// TIA Portal V17 export
// export: Created 2025-03-05T08:00:12.5882391Z, ExportSetting WithDefaults, DisplayName Totally Integrated Automation Portal, DisplayVersion V17 Update 8, DisplayName TIA Portal Openness, DisplayVersion V17 Update 8, DisplayName TIA Portal Version Control Interface, DisplayVersion V17, DisplayName SINAMICS Startdrive Advanced, DisplayVersion V17 SP2, DisplayName SINAMICS Startdrive G110M, G120, G120C, G120D, G120P, G115D, DisplayVersion V17 SP2, DisplayName SINAMICS Startdrive G130, G150, S120, S150, SINAMICS MV, S210, DisplayVersion V17 SP2, DisplayName STEP 7 Professional, DisplayVersion V17 Update 8, DisplayName SINUMERIK ONE STEP 7 Toolbox, DisplayVersion V17 Update 12, DisplayName SINUMERIK 840D sl STEP 7 Toolbox, DisplayVersion V17 Update 12, DisplayName STEP 7 Safety, DisplayVersion V17 Update 6, DisplayName WinCC Advanced, DisplayVersion V17 Update 8
FUNCTION "FC2121_MPP" : Void   // FC2121, LAD
{ S7_Optimized_Access := 'FALSE' }
AUTHOR : ETXETAR
VERSION : 1.0
// stored: AutoNumber false, IsIECCheckEnabled false, SetENOAutomatically false, UDAEnableTagReadback false
   VAR_TEMP
      ONE : Int;
      RETVAL1 : Int;
      SIMU_PANEL_HMI_SEL : Bool;   // SIMULATED PANEL IN HMI SELECTED
   END_VAR
   VAR CONSTANT
      FC_NUMBER : DInt := 2121;   // FC NUMBER
   END_VAR
   VAR_TEMP   // added for the SCL form of the ladder/FBD networks
      _w1 : Bool;
      _w2 : Bool;
   END_VAR
BEGIN

REGION Network 1: INPUTS
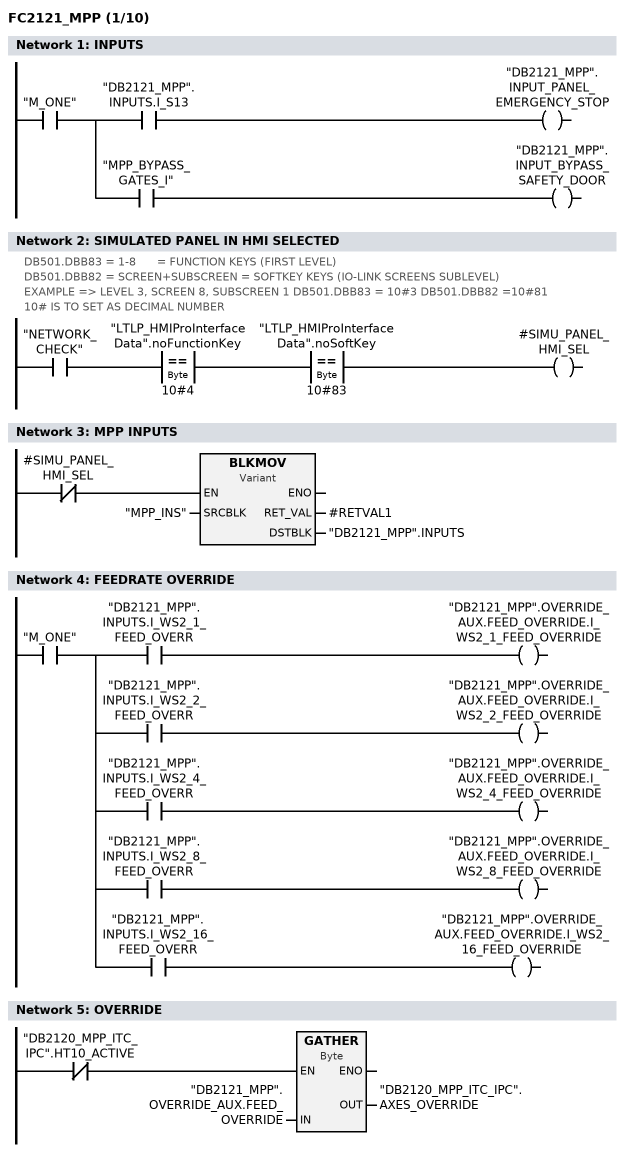
   RUNG wire#powerrail
      Contact( "M_ONE" )
      wire#w1
      Contact( "DB2121_MPP".INPUTS.I_S13 )
      Coil( "DB2121_MPP".INPUT_PANEL_EMERGENCY_STOP )
   END_RUNG
   RUNG wire#w1
      Contact( "MPP_BYPASS_GATES_I" )
      Coil( "DB2121_MPP".INPUT_BYPASS_SAFETY_DOOR )
   END_RUNG
   // the same network as SCL:
   "DB2121_MPP".INPUT_PANEL_EMERGENCY_STOP := "M_ONE" AND "DB2121_MPP".INPUTS.I_S13;
   "DB2121_MPP".INPUT_BYPASS_SAFETY_DOOR := "M_ONE" AND "MPP_BYPASS_GATES_I";
END_REGION

REGION Network 2: SIMULATED PANEL IN HMI SELECTED
   // DB501.DBB83 = 1-8      = FUNCTION KEYS (FIRST LEVEL)
   // DB501.DBB82 = SCREEN+SUBSCREEN = SOFTKEY KEYS (IO-LINK SCREENS SUBLEVEL)
   // EXAMPLE => LEVEL 3, SCREEN 8, SUBSCREEN 1 DB501.DBB83 = 10#3 DB501.DBB82 =10#81 
   // 10# IS TO SET AS DECIMAL NUMBER
   RUNG wire#powerrail
      Contact( "NETWORK_CHECK" )
      { S7_Templates := "SrcType := Byte" } EQ_Contact(in1 := "LTLP_HMIProInterfaceData".noFunctionKey, in2 := 10#4)
      { S7_Templates := "SrcType := Byte" } EQ_Contact(in1 := "LTLP_HMIProInterfaceData".noSoftKey, in2 := 10#83)
      Coil( #SIMU_PANEL_HMI_SEL )
   END_RUNG
   // the same network as SCL:
   #SIMU_PANEL_HMI_SEL := "NETWORK_CHECK" AND ("LTLP_HMIProInterfaceData".noFunctionKey = 10#4) AND ("LTLP_HMIProInterfaceData".noSoftKey = 10#83);
END_REGION

REGION Network 3: MPP INPUTS
   RUNG wire#powerrail
      I_Contact( #SIMU_PANEL_HMI_SEL )
      { S7_Templates := "blk_type := Variant" } BLKMOV(SRCBLK := "MPP_INS", RET_VAL => #RETVAL1, DSTBLK => "DB2121_MPP".INPUTS)
   END_RUNG
   // the same network as SCL:
   IF NOT #SIMU_PANEL_HMI_SEL THEN
       #RETVAL1 := BLKMOV(SRCBLK := "MPP_INS", DSTBLK => "DB2121_MPP".INPUTS);
   END_IF;
END_REGION

REGION Network 4: FEEDRATE OVERRIDE
   RUNG wire#powerrail
      Contact( "M_ONE" )
      wire#w1
      Contact( "DB2121_MPP".INPUTS.I_WS2_1_FEED_OVERR )
      Coil( "DB2121_MPP".OVERRIDE_AUX.FEED_OVERRIDE.I_WS2_1_FEED_OVERRIDE )
   END_RUNG
   RUNG wire#w1
      Contact( "DB2121_MPP".INPUTS.I_WS2_2_FEED_OVERR )
      Coil( "DB2121_MPP".OVERRIDE_AUX.FEED_OVERRIDE.I_WS2_2_FEED_OVERRIDE )
   END_RUNG
   RUNG wire#w1
      Contact( "DB2121_MPP".INPUTS.I_WS2_4_FEED_OVERR )
      Coil( "DB2121_MPP".OVERRIDE_AUX.FEED_OVERRIDE.I_WS2_4_FEED_OVERRIDE )
   END_RUNG
   RUNG wire#w1
      Contact( "DB2121_MPP".INPUTS.I_WS2_8_FEED_OVERR )
      Coil( "DB2121_MPP".OVERRIDE_AUX.FEED_OVERRIDE.I_WS2_8_FEED_OVERRIDE )
   END_RUNG
   RUNG wire#w1
      Contact( "DB2121_MPP".INPUTS.I_WS2_16_FEED_OVERR )
      Coil( "DB2121_MPP".OVERRIDE_AUX.FEED_OVERRIDE.I_WS2_16_FEED_OVERRIDE )
   END_RUNG
   // the same network as SCL:
   "DB2121_MPP".OVERRIDE_AUX.FEED_OVERRIDE.I_WS2_1_FEED_OVERRIDE := "M_ONE" AND "DB2121_MPP".INPUTS.I_WS2_1_FEED_OVERR;
   "DB2121_MPP".OVERRIDE_AUX.FEED_OVERRIDE.I_WS2_2_FEED_OVERRIDE := "M_ONE" AND "DB2121_MPP".INPUTS.I_WS2_2_FEED_OVERR;
   "DB2121_MPP".OVERRIDE_AUX.FEED_OVERRIDE.I_WS2_4_FEED_OVERRIDE := "M_ONE" AND "DB2121_MPP".INPUTS.I_WS2_4_FEED_OVERR;
   "DB2121_MPP".OVERRIDE_AUX.FEED_OVERRIDE.I_WS2_8_FEED_OVERRIDE := "M_ONE" AND "DB2121_MPP".INPUTS.I_WS2_8_FEED_OVERR;
   "DB2121_MPP".OVERRIDE_AUX.FEED_OVERRIDE.I_WS2_16_FEED_OVERRIDE := "M_ONE" AND "DB2121_MPP".INPUTS.I_WS2_16_FEED_OVERR;
END_REGION

REGION Network 5: OVERRIDE
   RUNG wire#powerrail
      I_Contact( "DB2120_MPP_ITC_IPC".HT10_ACTIVE )
      { S7_Templates := "[dest_type := Byte, src_type := Bool]" } GATHER(IN := "DB2121_MPP".OVERRIDE_AUX.FEED_OVERRIDE, OUT => "DB2120_MPP_ITC_IPC".AXES_OVERRIDE)
   END_RUNG
   // the same network as SCL:
   IF NOT "DB2120_MPP_ITC_IPC".HT10_ACTIVE THEN
       GATHER(IN := "DB2121_MPP".OVERRIDE_AUX.FEED_OVERRIDE, OUT => "DB2120_MPP_ITC_IPC".AXES_OVERRIDE);
   END_IF;
END_REGION

REGION Network 6: SPINDLES OVERRIDE
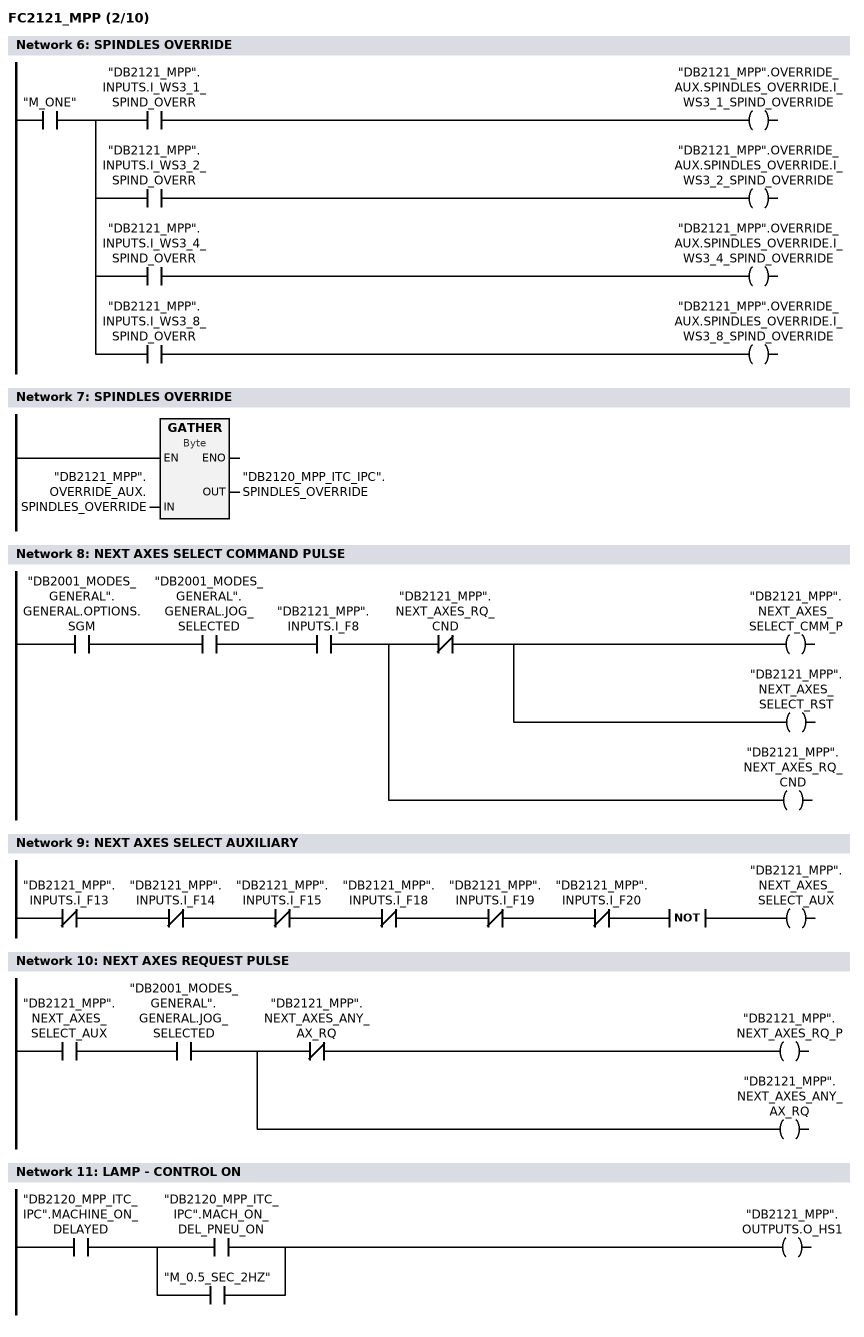
   RUNG wire#powerrail
      Contact( "M_ONE" )
      wire#w1
      Contact( "DB2121_MPP".INPUTS.I_WS3_1_SPIND_OVERR )
      Coil( "DB2121_MPP".OVERRIDE_AUX.SPINDLES_OVERRIDE.I_WS3_1_SPIND_OVERRIDE )
   END_RUNG
   RUNG wire#w1
      Contact( "DB2121_MPP".INPUTS.I_WS3_2_SPIND_OVERR )
      Coil( "DB2121_MPP".OVERRIDE_AUX.SPINDLES_OVERRIDE.I_WS3_2_SPIND_OVERRIDE )
   END_RUNG
   RUNG wire#w1
      Contact( "DB2121_MPP".INPUTS.I_WS3_4_SPIND_OVERR )
      Coil( "DB2121_MPP".OVERRIDE_AUX.SPINDLES_OVERRIDE.I_WS3_4_SPIND_OVERRIDE )
   END_RUNG
   RUNG wire#w1
      Contact( "DB2121_MPP".INPUTS.I_WS3_8_SPIND_OVERR )
      Coil( "DB2121_MPP".OVERRIDE_AUX.SPINDLES_OVERRIDE.I_WS3_8_SPIND_OVERRIDE )
   END_RUNG
   // the same network as SCL:
   "DB2121_MPP".OVERRIDE_AUX.SPINDLES_OVERRIDE.I_WS3_1_SPIND_OVERRIDE := "M_ONE" AND "DB2121_MPP".INPUTS.I_WS3_1_SPIND_OVERR;
   "DB2121_MPP".OVERRIDE_AUX.SPINDLES_OVERRIDE.I_WS3_2_SPIND_OVERRIDE := "M_ONE" AND "DB2121_MPP".INPUTS.I_WS3_2_SPIND_OVERR;
   "DB2121_MPP".OVERRIDE_AUX.SPINDLES_OVERRIDE.I_WS3_4_SPIND_OVERRIDE := "M_ONE" AND "DB2121_MPP".INPUTS.I_WS3_4_SPIND_OVERR;
   "DB2121_MPP".OVERRIDE_AUX.SPINDLES_OVERRIDE.I_WS3_8_SPIND_OVERRIDE := "M_ONE" AND "DB2121_MPP".INPUTS.I_WS3_8_SPIND_OVERR;
END_REGION

REGION Network 7: SPINDLES OVERRIDE
   RUNG wire#powerrail
      { S7_Templates := "[dest_type := Byte, src_type := Bool]" } GATHER(IN := "DB2121_MPP".OVERRIDE_AUX.SPINDLES_OVERRIDE, OUT => "DB2120_MPP_ITC_IPC".SPINDLES_OVERRIDE)
   END_RUNG
   // the same network as SCL:
   GATHER(IN := "DB2121_MPP".OVERRIDE_AUX.SPINDLES_OVERRIDE, OUT => "DB2120_MPP_ITC_IPC".SPINDLES_OVERRIDE);
END_REGION

REGION Network 8: NEXT AXES SELECT COMMAND PULSE
   RUNG wire#powerrail
      Contact( "DB2001_MODES_GENERAL".GENERAL.OPTIONS.SGM )
      Contact( "DB2001_MODES_GENERAL".GENERAL.JOG_SELECTED )
      Contact( "DB2121_MPP".INPUTS.I_F8 )
      wire#w1
      I_Contact( "DB2121_MPP".NEXT_AXES_RQ_CND )
      wire#w2
      Coil( "DB2121_MPP".NEXT_AXES_SELECT_CMM_P )
   END_RUNG
   RUNG wire#w2
      Coil( "DB2121_MPP".NEXT_AXES_SELECT_RST )
   END_RUNG
   RUNG wire#w1
      Coil( "DB2121_MPP".NEXT_AXES_RQ_CND )
   END_RUNG
   // the same network as SCL:
   #_w1 := "DB2001_MODES_GENERAL".GENERAL.OPTIONS.SGM AND "DB2001_MODES_GENERAL".GENERAL.JOG_SELECTED AND "DB2121_MPP".INPUTS.I_F8;
   "DB2121_MPP".NEXT_AXES_SELECT_CMM_P := #_w1 AND NOT "DB2121_MPP".NEXT_AXES_RQ_CND;
   "DB2121_MPP".NEXT_AXES_SELECT_RST := "DB2121_MPP".NEXT_AXES_SELECT_CMM_P;
   "DB2121_MPP".NEXT_AXES_RQ_CND := #_w1;
END_REGION

REGION Network 9: NEXT AXES SELECT AUXILIARY
   RUNG wire#powerrail
      I_Contact( "DB2121_MPP".INPUTS.I_F13 )
      I_Contact( "DB2121_MPP".INPUTS.I_F14 )
      I_Contact( "DB2121_MPP".INPUTS.I_F15 )
      I_Contact( "DB2121_MPP".INPUTS.I_F18 )
      I_Contact( "DB2121_MPP".INPUTS.I_F19 )
      I_Contact( "DB2121_MPP".INPUTS.I_F20 )
      Not()
      Coil( "DB2121_MPP".NEXT_AXES_SELECT_AUX )
   END_RUNG
   // the same network as SCL:
   "DB2121_MPP".NEXT_AXES_SELECT_AUX := NOT (NOT "DB2121_MPP".INPUTS.I_F13 AND NOT "DB2121_MPP".INPUTS.I_F14 AND NOT "DB2121_MPP".INPUTS.I_F15 AND NOT "DB2121_MPP".INPUTS.I_F18 AND NOT "DB2121_MPP".INPUTS.I_F19 AND NOT "DB2121_MPP".INPUTS.I_F20);
END_REGION

REGION Network 10: NEXT AXES REQUEST PULSE
   RUNG wire#powerrail
      Contact( "DB2121_MPP".NEXT_AXES_SELECT_AUX )
      Contact( "DB2001_MODES_GENERAL".GENERAL.JOG_SELECTED )
      wire#w1
      I_Contact( "DB2121_MPP".NEXT_AXES_ANY_AX_RQ )
      Coil( "DB2121_MPP".NEXT_AXES_RQ_P )
   END_RUNG
   RUNG wire#w1
      Coil( "DB2121_MPP".NEXT_AXES_ANY_AX_RQ )
   END_RUNG
   // the same network as SCL:
   #_w1 := "DB2121_MPP".NEXT_AXES_SELECT_AUX AND "DB2001_MODES_GENERAL".GENERAL.JOG_SELECTED;
   "DB2121_MPP".NEXT_AXES_RQ_P := #_w1 AND NOT "DB2121_MPP".NEXT_AXES_ANY_AX_RQ;
   "DB2121_MPP".NEXT_AXES_ANY_AX_RQ := #_w1;
END_REGION

REGION Network 11: LAMP - CONTROL ON
   RUNG wire#powerrail
      Contact( "DB2120_MPP_ITC_IPC".MACHINE_ON_DELAYED )
      wire#w1
      Contact( "DB2120_MPP_ITC_IPC".MACH_ON_DEL_PNEU_ON )
      wire#w2
      Coil( "DB2121_MPP".OUTPUTS.O_HS1 )
   END_RUNG
   RUNG wire#w1
      Contact( "M_0.5_SEC_2HZ" )
   END_RUNG wire#w2
   // the same network as SCL:
   "DB2121_MPP".OUTPUTS.O_HS1 := "DB2120_MPP_ITC_IPC".MACHINE_ON_DELAYED AND ("DB2120_MPP_ITC_IPC".MACH_ON_DEL_PNEU_ON OR "M_0.5_SEC_2HZ");
END_REGION

REGION Network 12: LAMP - HOME
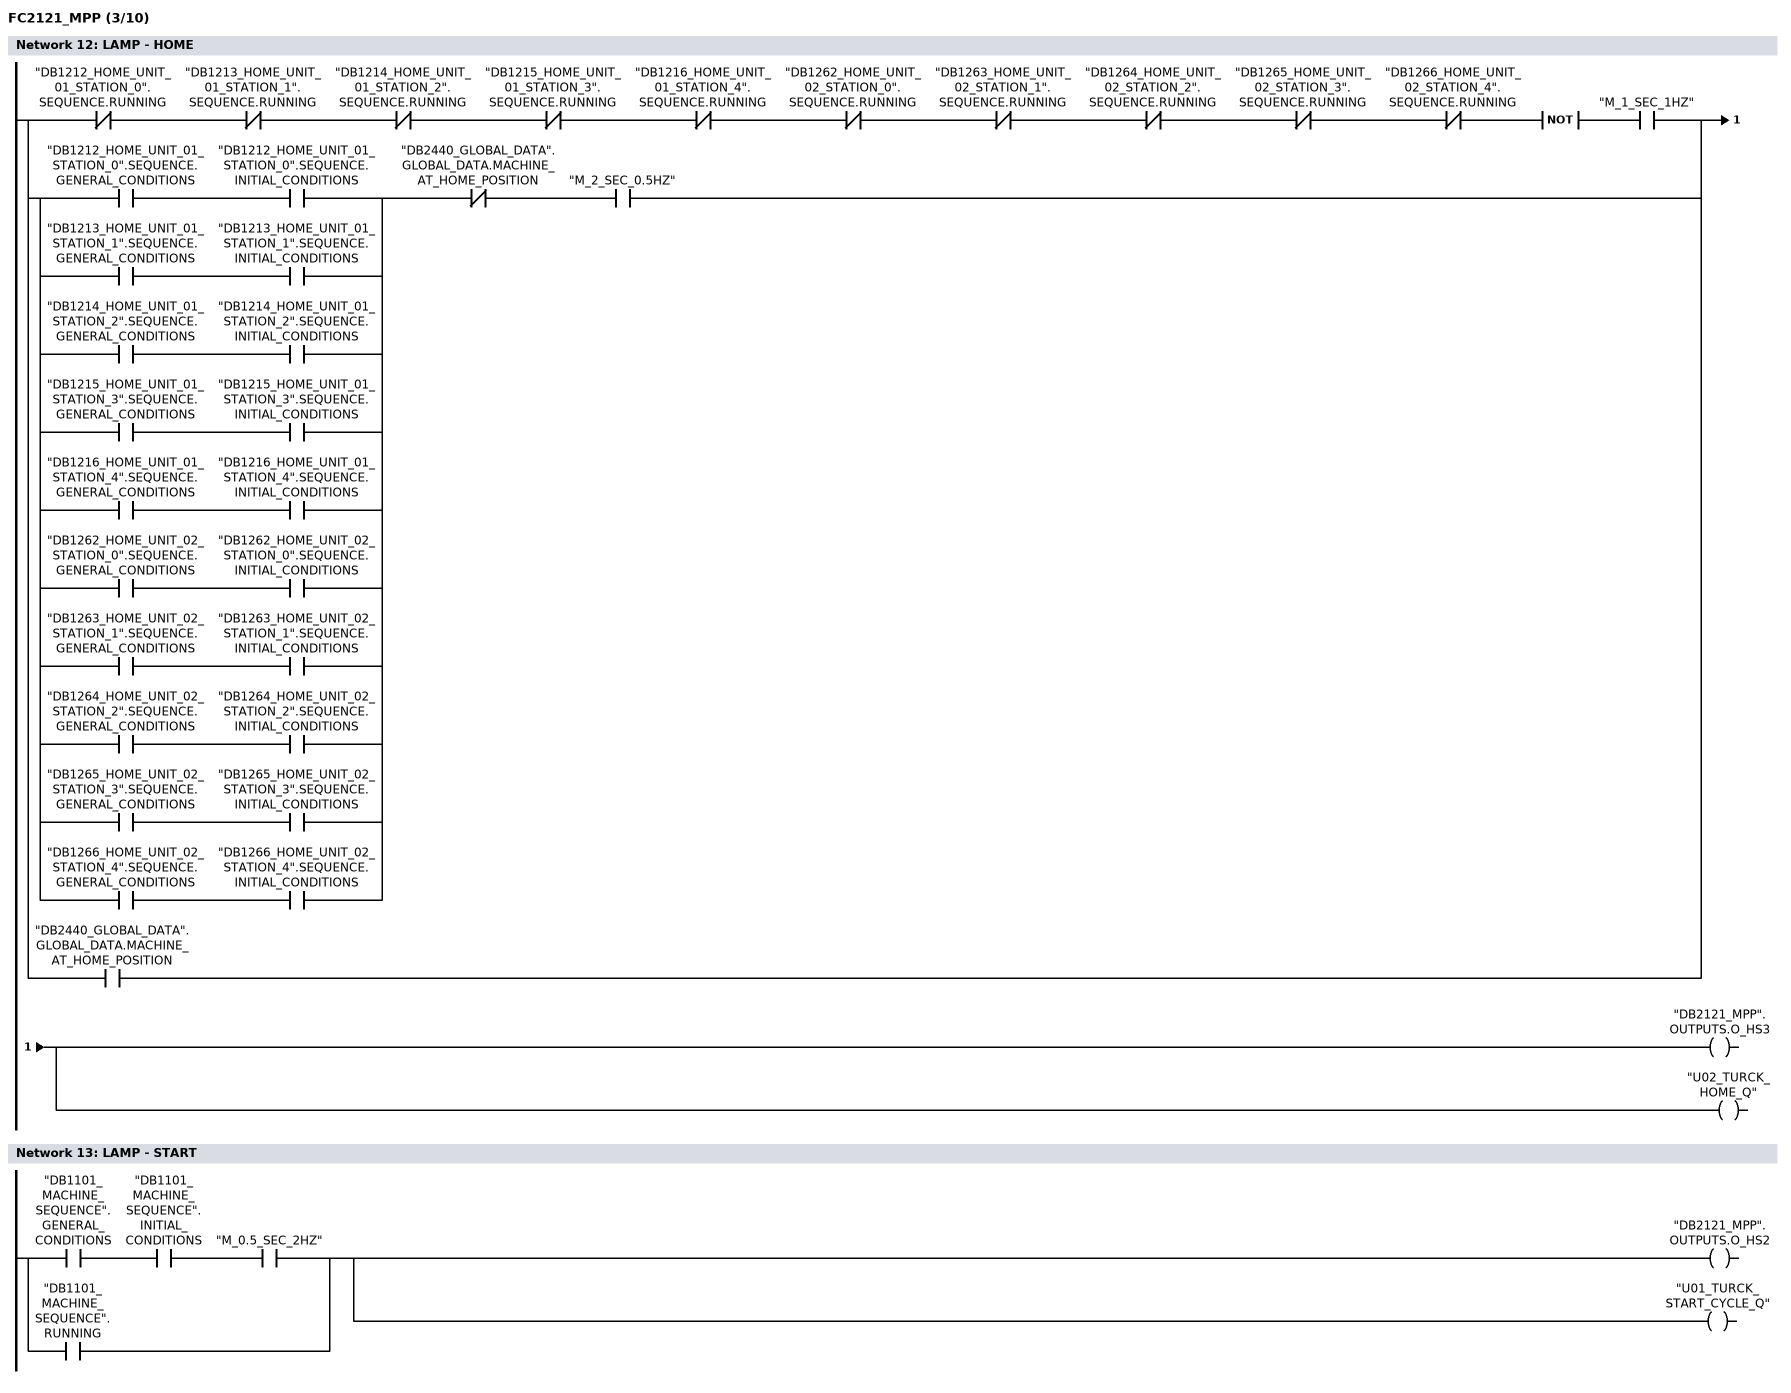
   RUNG wire#powerrail
      I_Contact( "DB1212_HOME_UNIT_01_STATION_0".SEQUENCE.RUNNING )
      I_Contact( "DB1213_HOME_UNIT_01_STATION_1".SEQUENCE.RUNNING )
      I_Contact( "DB1214_HOME_UNIT_01_STATION_2".SEQUENCE.RUNNING )
      I_Contact( "DB1215_HOME_UNIT_01_STATION_3".SEQUENCE.RUNNING )
      I_Contact( "DB1216_HOME_UNIT_01_STATION_4".SEQUENCE.RUNNING )
      I_Contact( "DB1262_HOME_UNIT_02_STATION_0".SEQUENCE.RUNNING )
      I_Contact( "DB1263_HOME_UNIT_02_STATION_1".SEQUENCE.RUNNING )
      I_Contact( "DB1264_HOME_UNIT_02_STATION_2".SEQUENCE.RUNNING )
      I_Contact( "DB1265_HOME_UNIT_02_STATION_3".SEQUENCE.RUNNING )
      I_Contact( "DB1266_HOME_UNIT_02_STATION_4".SEQUENCE.RUNNING )
      Not()
      Contact( "M_1_SEC_1HZ" )
      wire#w1
      Coil( "DB2121_MPP".OUTPUTS.O_HS3 )
   END_RUNG
   RUNG wire#powerrail
      Contact( "DB1212_HOME_UNIT_01_STATION_0".SEQUENCE.GENERAL_CONDITIONS )
      Contact( "DB1212_HOME_UNIT_01_STATION_0".SEQUENCE.INITIAL_CONDITIONS )
      wire#w2
      I_Contact( "DB2440_GLOBAL_DATA".GLOBAL_DATA.MACHINE_AT_HOME_POSITION )
      Contact( "M_2_SEC_0.5HZ" )
   END_RUNG wire#w1
   RUNG wire#powerrail
      Contact( "DB1213_HOME_UNIT_01_STATION_1".SEQUENCE.GENERAL_CONDITIONS )
      Contact( "DB1213_HOME_UNIT_01_STATION_1".SEQUENCE.INITIAL_CONDITIONS )
   END_RUNG wire#w2
   RUNG wire#powerrail
      Contact( "DB1214_HOME_UNIT_01_STATION_2".SEQUENCE.GENERAL_CONDITIONS )
      Contact( "DB1214_HOME_UNIT_01_STATION_2".SEQUENCE.INITIAL_CONDITIONS )
   END_RUNG wire#w2
   RUNG wire#powerrail
      Contact( "DB1215_HOME_UNIT_01_STATION_3".SEQUENCE.GENERAL_CONDITIONS )
      Contact( "DB1215_HOME_UNIT_01_STATION_3".SEQUENCE.INITIAL_CONDITIONS )
   END_RUNG wire#w2
   RUNG wire#powerrail
      Contact( "DB1216_HOME_UNIT_01_STATION_4".SEQUENCE.GENERAL_CONDITIONS )
      Contact( "DB1216_HOME_UNIT_01_STATION_4".SEQUENCE.INITIAL_CONDITIONS )
   END_RUNG wire#w2
   RUNG wire#powerrail
      Contact( "DB1262_HOME_UNIT_02_STATION_0".SEQUENCE.GENERAL_CONDITIONS )
      Contact( "DB1262_HOME_UNIT_02_STATION_0".SEQUENCE.INITIAL_CONDITIONS )
   END_RUNG wire#w2
   RUNG wire#powerrail
      Contact( "DB1263_HOME_UNIT_02_STATION_1".SEQUENCE.GENERAL_CONDITIONS )
      Contact( "DB1263_HOME_UNIT_02_STATION_1".SEQUENCE.INITIAL_CONDITIONS )
   END_RUNG wire#w2
   RUNG wire#powerrail
      Contact( "DB1264_HOME_UNIT_02_STATION_2".SEQUENCE.GENERAL_CONDITIONS )
      Contact( "DB1264_HOME_UNIT_02_STATION_2".SEQUENCE.INITIAL_CONDITIONS )
   END_RUNG wire#w2
   RUNG wire#powerrail
      Contact( "DB1265_HOME_UNIT_02_STATION_3".SEQUENCE.GENERAL_CONDITIONS )
      Contact( "DB1265_HOME_UNIT_02_STATION_3".SEQUENCE.INITIAL_CONDITIONS )
   END_RUNG wire#w2
   RUNG wire#powerrail
      Contact( "DB1266_HOME_UNIT_02_STATION_4".SEQUENCE.GENERAL_CONDITIONS )
      Contact( "DB1266_HOME_UNIT_02_STATION_4".SEQUENCE.INITIAL_CONDITIONS )
   END_RUNG wire#w2
   RUNG wire#powerrail
      Contact( "DB2440_GLOBAL_DATA".GLOBAL_DATA.MACHINE_AT_HOME_POSITION )
   END_RUNG wire#w1
   RUNG wire#w1
      Coil( "U02_TURCK_HOME_Q" )
   END_RUNG
   // the same network as SCL:
   "DB2121_MPP".OUTPUTS.O_HS3 := (NOT (NOT "DB1212_HOME_UNIT_01_STATION_0".SEQUENCE.RUNNING AND NOT "DB1213_HOME_UNIT_01_STATION_1".SEQUENCE.RUNNING AND NOT "DB1214_HOME_UNIT_01_STATION_2".SEQUENCE.RUNNING AND NOT "DB1215_HOME_UNIT_01_STATION_3".SEQUENCE.RUNNING AND NOT "DB1216_HOME_UNIT_01_STATION_4".SEQUENCE.RUNNING AND NOT "DB1262_HOME_UNIT_02_STATION_0".SEQUENCE.RUNNING AND NOT "DB1263_HOME_UNIT_02_STATION_1".SEQUENCE.RUNNING AND NOT "DB1264_HOME_UNIT_02_STATION_2".SEQUENCE.RUNNING AND NOT "DB1265_HOME_UNIT_02_STATION_3".SEQUENCE.RUNNING AND NOT "DB1266_HOME_UNIT_02_STATION_4".SEQUENCE.RUNNING) AND "M_1_SEC_1HZ") OR ((("DB1212_HOME_UNIT_01_STATION_0".SEQUENCE.GENERAL_CONDITIONS AND "DB1212_HOME_UNIT_01_STATION_0".SEQUENCE.INITIAL_CONDITIONS) OR ("DB1213_HOME_UNIT_01_STATION_1".SEQUENCE.GENERAL_CONDITIONS AND "DB1213_HOME_UNIT_01_STATION_1".SEQUENCE.INITIAL_CONDITIONS) OR ("DB1214_HOME_UNIT_01_STATION_2".SEQUENCE.GENERAL_CONDITIONS AND "DB1214_HOME_UNIT_01_STATION_2".SEQUENCE.INITIAL_CONDITIONS) OR ("DB1215_HOME_UNIT_01_STATION_3".SEQUENCE.GENERAL_CONDITIONS AND "DB1215_HOME_UNIT_01_STATION_3".SEQUENCE.INITIAL_CONDITIONS) OR ("DB1216_HOME_UNIT_01_STATION_4".SEQUENCE.GENERAL_CONDITIONS AND "DB1216_HOME_UNIT_01_STATION_4".SEQUENCE.INITIAL_CONDITIONS) OR ("DB1262_HOME_UNIT_02_STATION_0".SEQUENCE.GENERAL_CONDITIONS AND "DB1262_HOME_UNIT_02_STATION_0".SEQUENCE.INITIAL_CONDITIONS) OR ("DB1263_HOME_UNIT_02_STATION_1".SEQUENCE.GENERAL_CONDITIONS AND "DB1263_HOME_UNIT_02_STATION_1".SEQUENCE.INITIAL_CONDITIONS) OR ("DB1264_HOME_UNIT_02_STATION_2".SEQUENCE.GENERAL_CONDITIONS AND "DB1264_HOME_UNIT_02_STATION_2".SEQUENCE.INITIAL_CONDITIONS) OR ("DB1265_HOME_UNIT_02_STATION_3".SEQUENCE.GENERAL_CONDITIONS AND "DB1265_HOME_UNIT_02_STATION_3".SEQUENCE.INITIAL_CONDITIONS) OR ("DB1266_HOME_UNIT_02_STATION_4".SEQUENCE.GENERAL_CONDITIONS AND "DB1266_HOME_UNIT_02_STATION_4".SEQUENCE.INITIAL_CONDITIONS)) AND NOT "DB2440_GLOBAL_DATA".GLOBAL_DATA.MACHINE_AT_HOME_POSITION AND "M_2_SEC_0.5HZ") OR "DB2440_GLOBAL_DATA".GLOBAL_DATA.MACHINE_AT_HOME_POSITION;
   "U02_TURCK_HOME_Q" := "DB2121_MPP".OUTPUTS.O_HS3;
END_REGION

REGION Network 13: LAMP - START
   RUNG wire#powerrail
      Contact( "DB1101_MACHINE_SEQUENCE".GENERAL_CONDITIONS )
      Contact( "DB1101_MACHINE_SEQUENCE".INITIAL_CONDITIONS )
      Contact( "M_0.5_SEC_2HZ" )
      wire#w1
      Coil( "DB2121_MPP".OUTPUTS.O_HS2 )
   END_RUNG
   RUNG wire#powerrail
      Contact( "DB1101_MACHINE_SEQUENCE".RUNNING )
   END_RUNG wire#w1
   RUNG wire#w1
      Coil( "U01_TURCK_START_CYCLE_Q" )
   END_RUNG
   // the same network as SCL:
   "DB2121_MPP".OUTPUTS.O_HS2 := ("DB1101_MACHINE_SEQUENCE".GENERAL_CONDITIONS AND "DB1101_MACHINE_SEQUENCE".INITIAL_CONDITIONS AND "M_0.5_SEC_2HZ") OR "DB1101_MACHINE_SEQUENCE".RUNNING;
   "U01_TURCK_START_CYCLE_Q" := "DB2121_MPP".OUTPUTS.O_HS2;
END_REGION

REGION Network 14: LAMP - RESET FAULT
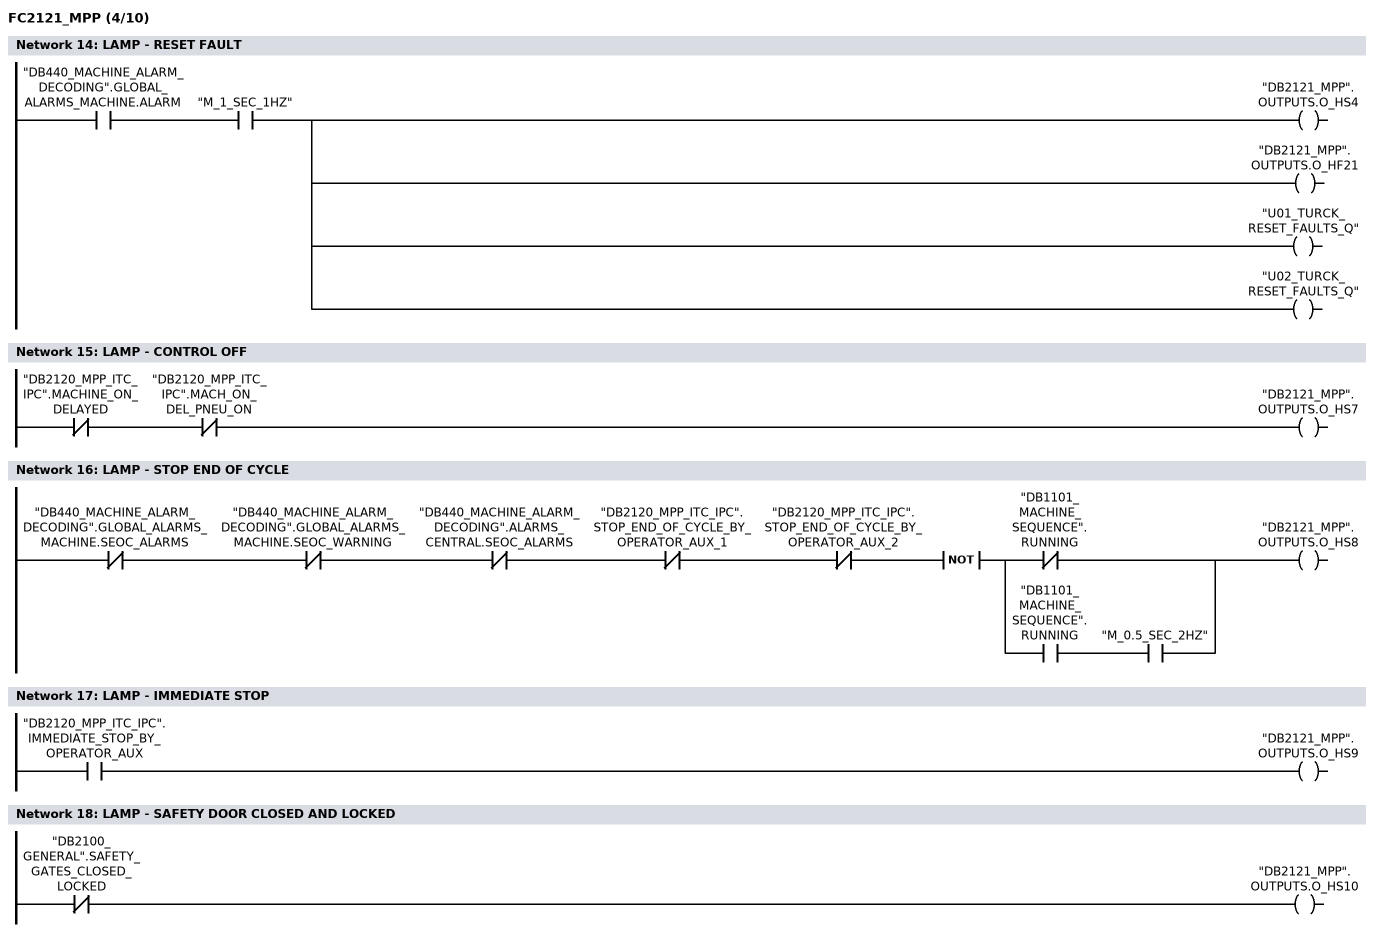
   RUNG wire#powerrail
      Contact( "DB440_MACHINE_ALARM_DECODING".GLOBAL_ALARMS_MACHINE.ALARM )
      Contact( "M_1_SEC_1HZ" )
      wire#w1
      Coil( "DB2121_MPP".OUTPUTS.O_HS4 )
   END_RUNG
   RUNG wire#w1
      Coil( "DB2121_MPP".OUTPUTS.O_HF21 )
   END_RUNG
   RUNG wire#w1
      Coil( "U01_TURCK_RESET_FAULTS_Q" )
   END_RUNG
   RUNG wire#w1
      Coil( "U02_TURCK_RESET_FAULTS_Q" )
   END_RUNG
   // the same network as SCL:
   "DB2121_MPP".OUTPUTS.O_HS4 := "DB440_MACHINE_ALARM_DECODING".GLOBAL_ALARMS_MACHINE.ALARM AND "M_1_SEC_1HZ";
   "DB2121_MPP".OUTPUTS.O_HF21 := "DB2121_MPP".OUTPUTS.O_HS4;
   "U01_TURCK_RESET_FAULTS_Q" := "DB2121_MPP".OUTPUTS.O_HS4;
   "U02_TURCK_RESET_FAULTS_Q" := "DB2121_MPP".OUTPUTS.O_HS4;
END_REGION

REGION Network 15: LAMP - CONTROL OFF
   RUNG wire#powerrail
      I_Contact( "DB2120_MPP_ITC_IPC".MACHINE_ON_DELAYED )
      I_Contact( "DB2120_MPP_ITC_IPC".MACH_ON_DEL_PNEU_ON )
      Coil( "DB2121_MPP".OUTPUTS.O_HS7 )
   END_RUNG
   // the same network as SCL:
   "DB2121_MPP".OUTPUTS.O_HS7 := NOT "DB2120_MPP_ITC_IPC".MACHINE_ON_DELAYED AND NOT "DB2120_MPP_ITC_IPC".MACH_ON_DEL_PNEU_ON;
END_REGION

REGION Network 16: LAMP - STOP END OF CYCLE
   RUNG wire#powerrail
      I_Contact( "DB440_MACHINE_ALARM_DECODING".GLOBAL_ALARMS_MACHINE.SEOC_ALARMS )
      I_Contact( "DB440_MACHINE_ALARM_DECODING".GLOBAL_ALARMS_MACHINE.SEOC_WARNING )
      I_Contact( "DB440_MACHINE_ALARM_DECODING".ALARMS_CENTRAL.SEOC_ALARMS )
      I_Contact( "DB2120_MPP_ITC_IPC".STOP_END_OF_CYCLE_BY_OPERATOR_AUX_1 )
      I_Contact( "DB2120_MPP_ITC_IPC".STOP_END_OF_CYCLE_BY_OPERATOR_AUX_2 )
      Not()
      wire#w1
      I_Contact( "DB1101_MACHINE_SEQUENCE".RUNNING )
      wire#w2
      Coil( "DB2121_MPP".OUTPUTS.O_HS8 )
   END_RUNG
   RUNG wire#w1
      Contact( "DB1101_MACHINE_SEQUENCE".RUNNING )
      Contact( "M_0.5_SEC_2HZ" )
   END_RUNG wire#w2
   // the same network as SCL:
   "DB2121_MPP".OUTPUTS.O_HS8 := NOT (NOT "DB440_MACHINE_ALARM_DECODING".GLOBAL_ALARMS_MACHINE.SEOC_ALARMS AND NOT "DB440_MACHINE_ALARM_DECODING".GLOBAL_ALARMS_MACHINE.SEOC_WARNING AND NOT "DB440_MACHINE_ALARM_DECODING".ALARMS_CENTRAL.SEOC_ALARMS AND NOT "DB2120_MPP_ITC_IPC".STOP_END_OF_CYCLE_BY_OPERATOR_AUX_1 AND NOT "DB2120_MPP_ITC_IPC".STOP_END_OF_CYCLE_BY_OPERATOR_AUX_2) AND (NOT "DB1101_MACHINE_SEQUENCE".RUNNING OR ("DB1101_MACHINE_SEQUENCE".RUNNING AND "M_0.5_SEC_2HZ"));
END_REGION

REGION Network 17: LAMP - IMMEDIATE STOP
   RUNG wire#powerrail
      Contact( "DB2120_MPP_ITC_IPC".IMMEDIATE_STOP_BY_OPERATOR_AUX )
      Coil( "DB2121_MPP".OUTPUTS.O_HS9 )
   END_RUNG
   // the same network as SCL:
   "DB2121_MPP".OUTPUTS.O_HS9 := "DB2120_MPP_ITC_IPC".IMMEDIATE_STOP_BY_OPERATOR_AUX;
END_REGION

REGION Network 18: LAMP - SAFETY DOOR CLOSED AND LOCKED
   RUNG wire#powerrail
      I_Contact( "DB2100_GENERAL".SAFETY_GATES_CLOSED_LOCKED )
      Coil( "DB2121_MPP".OUTPUTS.O_HS10 )
   END_RUNG
   // the same network as SCL:
   "DB2121_MPP".OUTPUTS.O_HS10 := NOT "DB2100_GENERAL".SAFETY_GATES_CLOSED_LOCKED;
END_REGION

REGION Network 19: LAMP - MANUAL LOAD PART U01
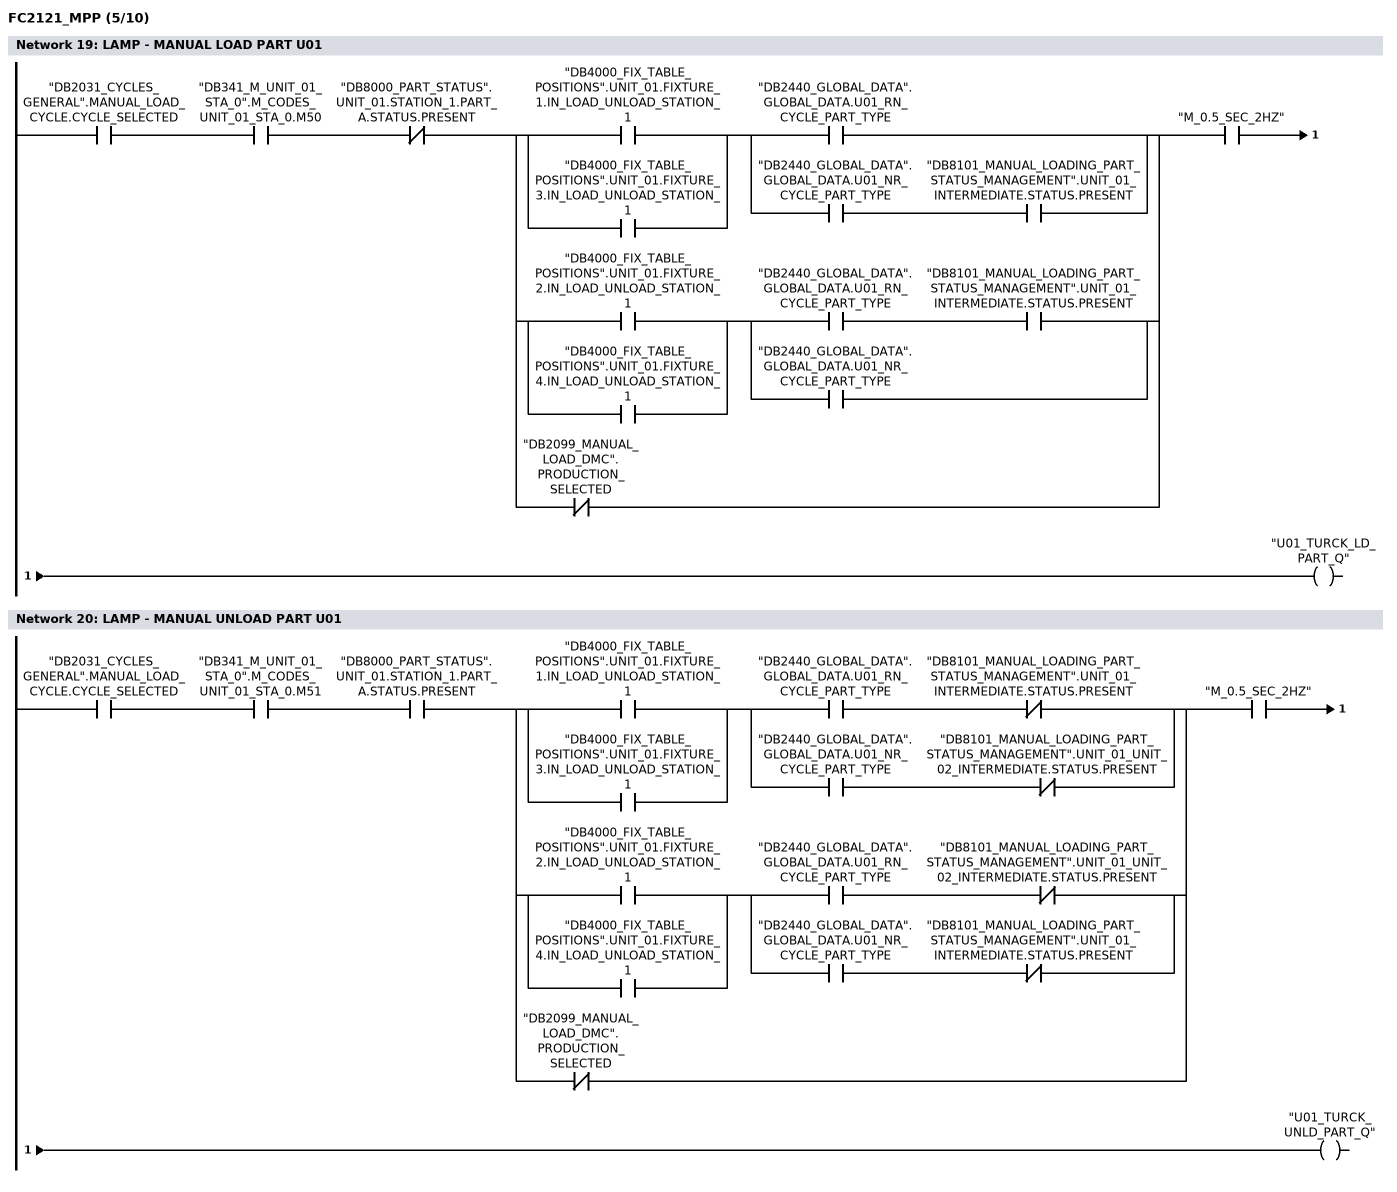
   RUNG wire#powerrail
      Contact( "DB2031_CYCLES_GENERAL".MANUAL_LOAD_CYCLE.CYCLE_SELECTED )
      Contact( "DB341_M_UNIT_01_STA_0".M_CODES_UNIT_01_STA_0.M50 )
      I_Contact( "DB8000_PART_STATUS".UNIT_01.STATION_1.PART_A.STATUS.PRESENT )
      wire#w1
      Contact( "DB4000_FIX_TABLE_POSITIONS".UNIT_01.FIXTURE_1.IN_LOAD_UNLOAD_STATION_1 )
      wire#w2
      Contact( "DB2440_GLOBAL_DATA".GLOBAL_DATA.U01_RN_CYCLE_PART_TYPE )
      wire#w3
      Contact( "M_0.5_SEC_2HZ" )
      Coil( "U01_TURCK_LD_PART_Q" )
   END_RUNG
   RUNG wire#w1
      Contact( "DB4000_FIX_TABLE_POSITIONS".UNIT_01.FIXTURE_3.IN_LOAD_UNLOAD_STATION_1 )
   END_RUNG wire#w2
   RUNG wire#w2
      Contact( "DB2440_GLOBAL_DATA".GLOBAL_DATA.U01_NR_CYCLE_PART_TYPE )
      Contact( "DB8101_MANUAL_LOADING_PART_STATUS_MANAGEMENT".UNIT_01_INTERMEDIATE.STATUS.PRESENT )
   END_RUNG wire#w3
   RUNG wire#w1
      Contact( "DB4000_FIX_TABLE_POSITIONS".UNIT_01.FIXTURE_2.IN_LOAD_UNLOAD_STATION_1 )
      wire#w4
      Contact( "DB2440_GLOBAL_DATA".GLOBAL_DATA.U01_RN_CYCLE_PART_TYPE )
      Contact( "DB8101_MANUAL_LOADING_PART_STATUS_MANAGEMENT".UNIT_01_INTERMEDIATE.STATUS.PRESENT )
   END_RUNG wire#w3
   RUNG wire#w1
      Contact( "DB4000_FIX_TABLE_POSITIONS".UNIT_01.FIXTURE_4.IN_LOAD_UNLOAD_STATION_1 )
   END_RUNG wire#w4
   RUNG wire#w4
      Contact( "DB2440_GLOBAL_DATA".GLOBAL_DATA.U01_NR_CYCLE_PART_TYPE )
   END_RUNG wire#w3
   RUNG wire#w1
      I_Contact( "DB2099_MANUAL_LOAD_DMC".PRODUCTION_SELECTED )
   END_RUNG wire#w3
   // the same network as SCL:
   "U01_TURCK_LD_PART_Q" := "DB2031_CYCLES_GENERAL".MANUAL_LOAD_CYCLE.CYCLE_SELECTED AND "DB341_M_UNIT_01_STA_0".M_CODES_UNIT_01_STA_0.M50 AND NOT "DB8000_PART_STATUS".UNIT_01.STATION_1.PART_A.STATUS.PRESENT AND ((("DB4000_FIX_TABLE_POSITIONS".UNIT_01.FIXTURE_1.IN_LOAD_UNLOAD_STATION_1 OR "DB4000_FIX_TABLE_POSITIONS".UNIT_01.FIXTURE_3.IN_LOAD_UNLOAD_STATION_1) AND ("DB2440_GLOBAL_DATA".GLOBAL_DATA.U01_RN_CYCLE_PART_TYPE OR ("DB2440_GLOBAL_DATA".GLOBAL_DATA.U01_NR_CYCLE_PART_TYPE AND "DB8101_MANUAL_LOADING_PART_STATUS_MANAGEMENT".UNIT_01_INTERMEDIATE.STATUS.PRESENT))) OR (("DB4000_FIX_TABLE_POSITIONS".UNIT_01.FIXTURE_2.IN_LOAD_UNLOAD_STATION_1 OR "DB4000_FIX_TABLE_POSITIONS".UNIT_01.FIXTURE_4.IN_LOAD_UNLOAD_STATION_1) AND (("DB2440_GLOBAL_DATA".GLOBAL_DATA.U01_RN_CYCLE_PART_TYPE AND "DB8101_MANUAL_LOADING_PART_STATUS_MANAGEMENT".UNIT_01_INTERMEDIATE.STATUS.PRESENT) OR "DB2440_GLOBAL_DATA".GLOBAL_DATA.U01_NR_CYCLE_PART_TYPE)) OR NOT "DB2099_MANUAL_LOAD_DMC".PRODUCTION_SELECTED) AND "M_0.5_SEC_2HZ";
END_REGION

REGION Network 20: LAMP - MANUAL UNLOAD PART U01
   RUNG wire#powerrail
      Contact( "DB2031_CYCLES_GENERAL".MANUAL_LOAD_CYCLE.CYCLE_SELECTED )
      Contact( "DB341_M_UNIT_01_STA_0".M_CODES_UNIT_01_STA_0.M51 )
      Contact( "DB8000_PART_STATUS".UNIT_01.STATION_1.PART_A.STATUS.PRESENT )
      wire#w1
      Contact( "DB4000_FIX_TABLE_POSITIONS".UNIT_01.FIXTURE_1.IN_LOAD_UNLOAD_STATION_1 )
      wire#w2
      Contact( "DB2440_GLOBAL_DATA".GLOBAL_DATA.U01_RN_CYCLE_PART_TYPE )
      I_Contact( "DB8101_MANUAL_LOADING_PART_STATUS_MANAGEMENT".UNIT_01_INTERMEDIATE.STATUS.PRESENT )
      wire#w3
      Contact( "M_0.5_SEC_2HZ" )
      Coil( "U01_TURCK_UNLD_PART_Q" )
   END_RUNG
   RUNG wire#w1
      Contact( "DB4000_FIX_TABLE_POSITIONS".UNIT_01.FIXTURE_3.IN_LOAD_UNLOAD_STATION_1 )
   END_RUNG wire#w2
   RUNG wire#w2
      Contact( "DB2440_GLOBAL_DATA".GLOBAL_DATA.U01_NR_CYCLE_PART_TYPE )
      I_Contact( "DB8101_MANUAL_LOADING_PART_STATUS_MANAGEMENT".UNIT_01_UNIT_02_INTERMEDIATE.STATUS.PRESENT )
   END_RUNG wire#w3
   RUNG wire#w1
      Contact( "DB4000_FIX_TABLE_POSITIONS".UNIT_01.FIXTURE_2.IN_LOAD_UNLOAD_STATION_1 )
      wire#w4
      Contact( "DB2440_GLOBAL_DATA".GLOBAL_DATA.U01_RN_CYCLE_PART_TYPE )
      I_Contact( "DB8101_MANUAL_LOADING_PART_STATUS_MANAGEMENT".UNIT_01_UNIT_02_INTERMEDIATE.STATUS.PRESENT )
   END_RUNG wire#w3
   RUNG wire#w1
      Contact( "DB4000_FIX_TABLE_POSITIONS".UNIT_01.FIXTURE_4.IN_LOAD_UNLOAD_STATION_1 )
   END_RUNG wire#w4
   RUNG wire#w4
      Contact( "DB2440_GLOBAL_DATA".GLOBAL_DATA.U01_NR_CYCLE_PART_TYPE )
      I_Contact( "DB8101_MANUAL_LOADING_PART_STATUS_MANAGEMENT".UNIT_01_INTERMEDIATE.STATUS.PRESENT )
   END_RUNG wire#w3
   RUNG wire#w1
      I_Contact( "DB2099_MANUAL_LOAD_DMC".PRODUCTION_SELECTED )
   END_RUNG wire#w3
   // the same network as SCL:
   "U01_TURCK_UNLD_PART_Q" := "DB2031_CYCLES_GENERAL".MANUAL_LOAD_CYCLE.CYCLE_SELECTED AND "DB341_M_UNIT_01_STA_0".M_CODES_UNIT_01_STA_0.M51 AND "DB8000_PART_STATUS".UNIT_01.STATION_1.PART_A.STATUS.PRESENT AND ((("DB4000_FIX_TABLE_POSITIONS".UNIT_01.FIXTURE_1.IN_LOAD_UNLOAD_STATION_1 OR "DB4000_FIX_TABLE_POSITIONS".UNIT_01.FIXTURE_3.IN_LOAD_UNLOAD_STATION_1) AND (("DB2440_GLOBAL_DATA".GLOBAL_DATA.U01_RN_CYCLE_PART_TYPE AND NOT "DB8101_MANUAL_LOADING_PART_STATUS_MANAGEMENT".UNIT_01_INTERMEDIATE.STATUS.PRESENT) OR ("DB2440_GLOBAL_DATA".GLOBAL_DATA.U01_NR_CYCLE_PART_TYPE AND NOT "DB8101_MANUAL_LOADING_PART_STATUS_MANAGEMENT".UNIT_01_UNIT_02_INTERMEDIATE.STATUS.PRESENT))) OR (("DB4000_FIX_TABLE_POSITIONS".UNIT_01.FIXTURE_2.IN_LOAD_UNLOAD_STATION_1 OR "DB4000_FIX_TABLE_POSITIONS".UNIT_01.FIXTURE_4.IN_LOAD_UNLOAD_STATION_1) AND (("DB2440_GLOBAL_DATA".GLOBAL_DATA.U01_RN_CYCLE_PART_TYPE AND NOT "DB8101_MANUAL_LOADING_PART_STATUS_MANAGEMENT".UNIT_01_UNIT_02_INTERMEDIATE.STATUS.PRESENT) OR ("DB2440_GLOBAL_DATA".GLOBAL_DATA.U01_NR_CYCLE_PART_TYPE AND NOT "DB8101_MANUAL_LOADING_PART_STATUS_MANAGEMENT".UNIT_01_INTERMEDIATE.STATUS.PRESENT))) OR NOT "DB2099_MANUAL_LOAD_DMC".PRODUCTION_SELECTED) AND "M_0.5_SEC_2HZ";
END_REGION

REGION Network 21: LAMP - MANUAL LOAD PART U02
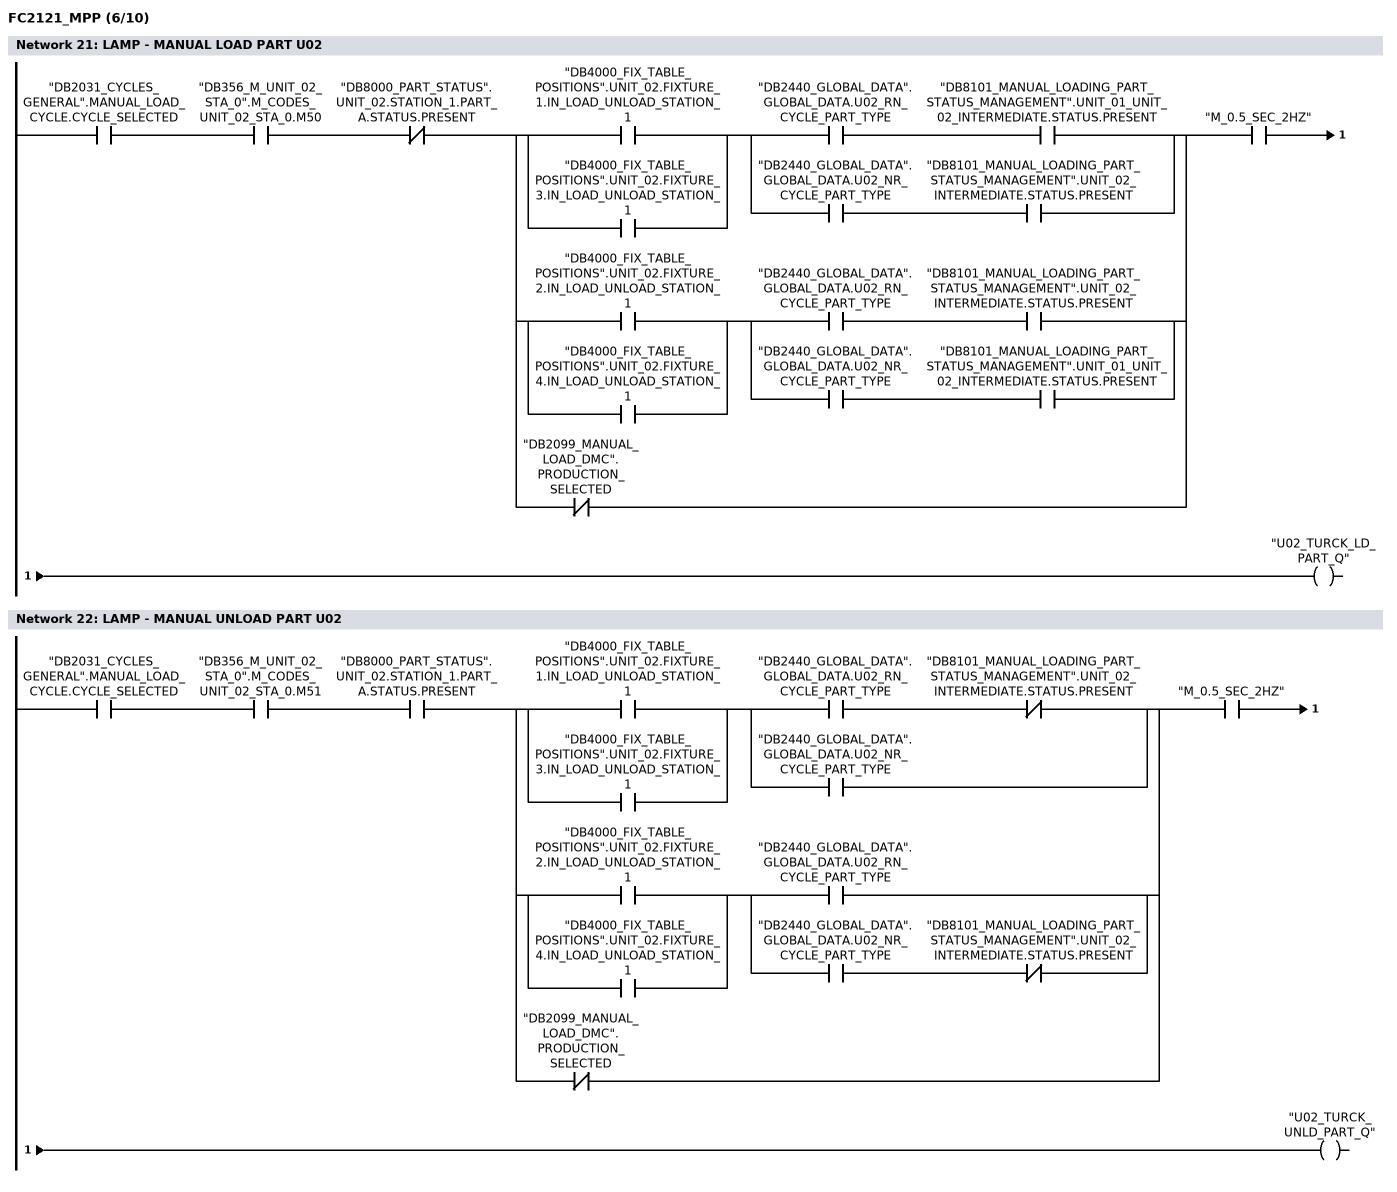
   RUNG wire#powerrail
      Contact( "DB2031_CYCLES_GENERAL".MANUAL_LOAD_CYCLE.CYCLE_SELECTED )
      Contact( "DB356_M_UNIT_02_STA_0".M_CODES_UNIT_02_STA_0.M50 )
      I_Contact( "DB8000_PART_STATUS".UNIT_02.STATION_1.PART_A.STATUS.PRESENT )
      wire#w1
      Contact( "DB4000_FIX_TABLE_POSITIONS".UNIT_02.FIXTURE_1.IN_LOAD_UNLOAD_STATION_1 )
      wire#w2
      Contact( "DB2440_GLOBAL_DATA".GLOBAL_DATA.U02_RN_CYCLE_PART_TYPE )
      Contact( "DB8101_MANUAL_LOADING_PART_STATUS_MANAGEMENT".UNIT_01_UNIT_02_INTERMEDIATE.STATUS.PRESENT )
      wire#w3
      Contact( "M_0.5_SEC_2HZ" )
      Coil( "U02_TURCK_LD_PART_Q" )
   END_RUNG
   RUNG wire#w1
      Contact( "DB4000_FIX_TABLE_POSITIONS".UNIT_02.FIXTURE_3.IN_LOAD_UNLOAD_STATION_1 )
   END_RUNG wire#w2
   RUNG wire#w2
      Contact( "DB2440_GLOBAL_DATA".GLOBAL_DATA.U02_NR_CYCLE_PART_TYPE )
      Contact( "DB8101_MANUAL_LOADING_PART_STATUS_MANAGEMENT".UNIT_02_INTERMEDIATE.STATUS.PRESENT )
   END_RUNG wire#w3
   RUNG wire#w1
      Contact( "DB4000_FIX_TABLE_POSITIONS".UNIT_02.FIXTURE_2.IN_LOAD_UNLOAD_STATION_1 )
      wire#w4
      Contact( "DB2440_GLOBAL_DATA".GLOBAL_DATA.U02_RN_CYCLE_PART_TYPE )
      Contact( "DB8101_MANUAL_LOADING_PART_STATUS_MANAGEMENT".UNIT_02_INTERMEDIATE.STATUS.PRESENT )
   END_RUNG wire#w3
   RUNG wire#w1
      Contact( "DB4000_FIX_TABLE_POSITIONS".UNIT_02.FIXTURE_4.IN_LOAD_UNLOAD_STATION_1 )
   END_RUNG wire#w4
   RUNG wire#w4
      Contact( "DB2440_GLOBAL_DATA".GLOBAL_DATA.U02_NR_CYCLE_PART_TYPE )
      Contact( "DB8101_MANUAL_LOADING_PART_STATUS_MANAGEMENT".UNIT_01_UNIT_02_INTERMEDIATE.STATUS.PRESENT )
   END_RUNG wire#w3
   RUNG wire#w1
      I_Contact( "DB2099_MANUAL_LOAD_DMC".PRODUCTION_SELECTED )
   END_RUNG wire#w3
   // the same network as SCL:
   "U02_TURCK_LD_PART_Q" := "DB2031_CYCLES_GENERAL".MANUAL_LOAD_CYCLE.CYCLE_SELECTED AND "DB356_M_UNIT_02_STA_0".M_CODES_UNIT_02_STA_0.M50 AND NOT "DB8000_PART_STATUS".UNIT_02.STATION_1.PART_A.STATUS.PRESENT AND ((("DB4000_FIX_TABLE_POSITIONS".UNIT_02.FIXTURE_1.IN_LOAD_UNLOAD_STATION_1 OR "DB4000_FIX_TABLE_POSITIONS".UNIT_02.FIXTURE_3.IN_LOAD_UNLOAD_STATION_1) AND (("DB2440_GLOBAL_DATA".GLOBAL_DATA.U02_RN_CYCLE_PART_TYPE AND "DB8101_MANUAL_LOADING_PART_STATUS_MANAGEMENT".UNIT_01_UNIT_02_INTERMEDIATE.STATUS.PRESENT) OR ("DB2440_GLOBAL_DATA".GLOBAL_DATA.U02_NR_CYCLE_PART_TYPE AND "DB8101_MANUAL_LOADING_PART_STATUS_MANAGEMENT".UNIT_02_INTERMEDIATE.STATUS.PRESENT))) OR (("DB4000_FIX_TABLE_POSITIONS".UNIT_02.FIXTURE_2.IN_LOAD_UNLOAD_STATION_1 OR "DB4000_FIX_TABLE_POSITIONS".UNIT_02.FIXTURE_4.IN_LOAD_UNLOAD_STATION_1) AND (("DB2440_GLOBAL_DATA".GLOBAL_DATA.U02_RN_CYCLE_PART_TYPE AND "DB8101_MANUAL_LOADING_PART_STATUS_MANAGEMENT".UNIT_02_INTERMEDIATE.STATUS.PRESENT) OR ("DB2440_GLOBAL_DATA".GLOBAL_DATA.U02_NR_CYCLE_PART_TYPE AND "DB8101_MANUAL_LOADING_PART_STATUS_MANAGEMENT".UNIT_01_UNIT_02_INTERMEDIATE.STATUS.PRESENT))) OR NOT "DB2099_MANUAL_LOAD_DMC".PRODUCTION_SELECTED) AND "M_0.5_SEC_2HZ";
END_REGION

REGION Network 22: LAMP - MANUAL UNLOAD PART U02
   RUNG wire#powerrail
      Contact( "DB2031_CYCLES_GENERAL".MANUAL_LOAD_CYCLE.CYCLE_SELECTED )
      Contact( "DB356_M_UNIT_02_STA_0".M_CODES_UNIT_02_STA_0.M51 )
      Contact( "DB8000_PART_STATUS".UNIT_02.STATION_1.PART_A.STATUS.PRESENT )
      wire#w1
      Contact( "DB4000_FIX_TABLE_POSITIONS".UNIT_02.FIXTURE_1.IN_LOAD_UNLOAD_STATION_1 )
      wire#w2
      Contact( "DB2440_GLOBAL_DATA".GLOBAL_DATA.U02_RN_CYCLE_PART_TYPE )
      I_Contact( "DB8101_MANUAL_LOADING_PART_STATUS_MANAGEMENT".UNIT_02_INTERMEDIATE.STATUS.PRESENT )
      wire#w3
      Contact( "M_0.5_SEC_2HZ" )
      Coil( "U02_TURCK_UNLD_PART_Q" )
   END_RUNG
   RUNG wire#w1
      Contact( "DB4000_FIX_TABLE_POSITIONS".UNIT_02.FIXTURE_3.IN_LOAD_UNLOAD_STATION_1 )
   END_RUNG wire#w2
   RUNG wire#w2
      Contact( "DB2440_GLOBAL_DATA".GLOBAL_DATA.U02_NR_CYCLE_PART_TYPE )
   END_RUNG wire#w3
   RUNG wire#w1
      Contact( "DB4000_FIX_TABLE_POSITIONS".UNIT_02.FIXTURE_2.IN_LOAD_UNLOAD_STATION_1 )
      wire#w4
      Contact( "DB2440_GLOBAL_DATA".GLOBAL_DATA.U02_RN_CYCLE_PART_TYPE )
   END_RUNG wire#w3
   RUNG wire#w1
      Contact( "DB4000_FIX_TABLE_POSITIONS".UNIT_02.FIXTURE_4.IN_LOAD_UNLOAD_STATION_1 )
   END_RUNG wire#w4
   RUNG wire#w4
      Contact( "DB2440_GLOBAL_DATA".GLOBAL_DATA.U02_NR_CYCLE_PART_TYPE )
      I_Contact( "DB8101_MANUAL_LOADING_PART_STATUS_MANAGEMENT".UNIT_02_INTERMEDIATE.STATUS.PRESENT )
   END_RUNG wire#w3
   RUNG wire#w1
      I_Contact( "DB2099_MANUAL_LOAD_DMC".PRODUCTION_SELECTED )
   END_RUNG wire#w3
   // the same network as SCL:
   "U02_TURCK_UNLD_PART_Q" := "DB2031_CYCLES_GENERAL".MANUAL_LOAD_CYCLE.CYCLE_SELECTED AND "DB356_M_UNIT_02_STA_0".M_CODES_UNIT_02_STA_0.M51 AND "DB8000_PART_STATUS".UNIT_02.STATION_1.PART_A.STATUS.PRESENT AND ((("DB4000_FIX_TABLE_POSITIONS".UNIT_02.FIXTURE_1.IN_LOAD_UNLOAD_STATION_1 OR "DB4000_FIX_TABLE_POSITIONS".UNIT_02.FIXTURE_3.IN_LOAD_UNLOAD_STATION_1) AND (("DB2440_GLOBAL_DATA".GLOBAL_DATA.U02_RN_CYCLE_PART_TYPE AND NOT "DB8101_MANUAL_LOADING_PART_STATUS_MANAGEMENT".UNIT_02_INTERMEDIATE.STATUS.PRESENT) OR "DB2440_GLOBAL_DATA".GLOBAL_DATA.U02_NR_CYCLE_PART_TYPE)) OR (("DB4000_FIX_TABLE_POSITIONS".UNIT_02.FIXTURE_2.IN_LOAD_UNLOAD_STATION_1 OR "DB4000_FIX_TABLE_POSITIONS".UNIT_02.FIXTURE_4.IN_LOAD_UNLOAD_STATION_1) AND ("DB2440_GLOBAL_DATA".GLOBAL_DATA.U02_RN_CYCLE_PART_TYPE OR ("DB2440_GLOBAL_DATA".GLOBAL_DATA.U02_NR_CYCLE_PART_TYPE AND NOT "DB8101_MANUAL_LOADING_PART_STATUS_MANAGEMENT".UNIT_02_INTERMEDIATE.STATUS.PRESENT))) OR NOT "DB2099_MANUAL_LOAD_DMC".PRODUCTION_SELECTED) AND "M_0.5_SEC_2HZ";
END_REGION

REGION Network 23: MPP HF LAMPS CYCLES
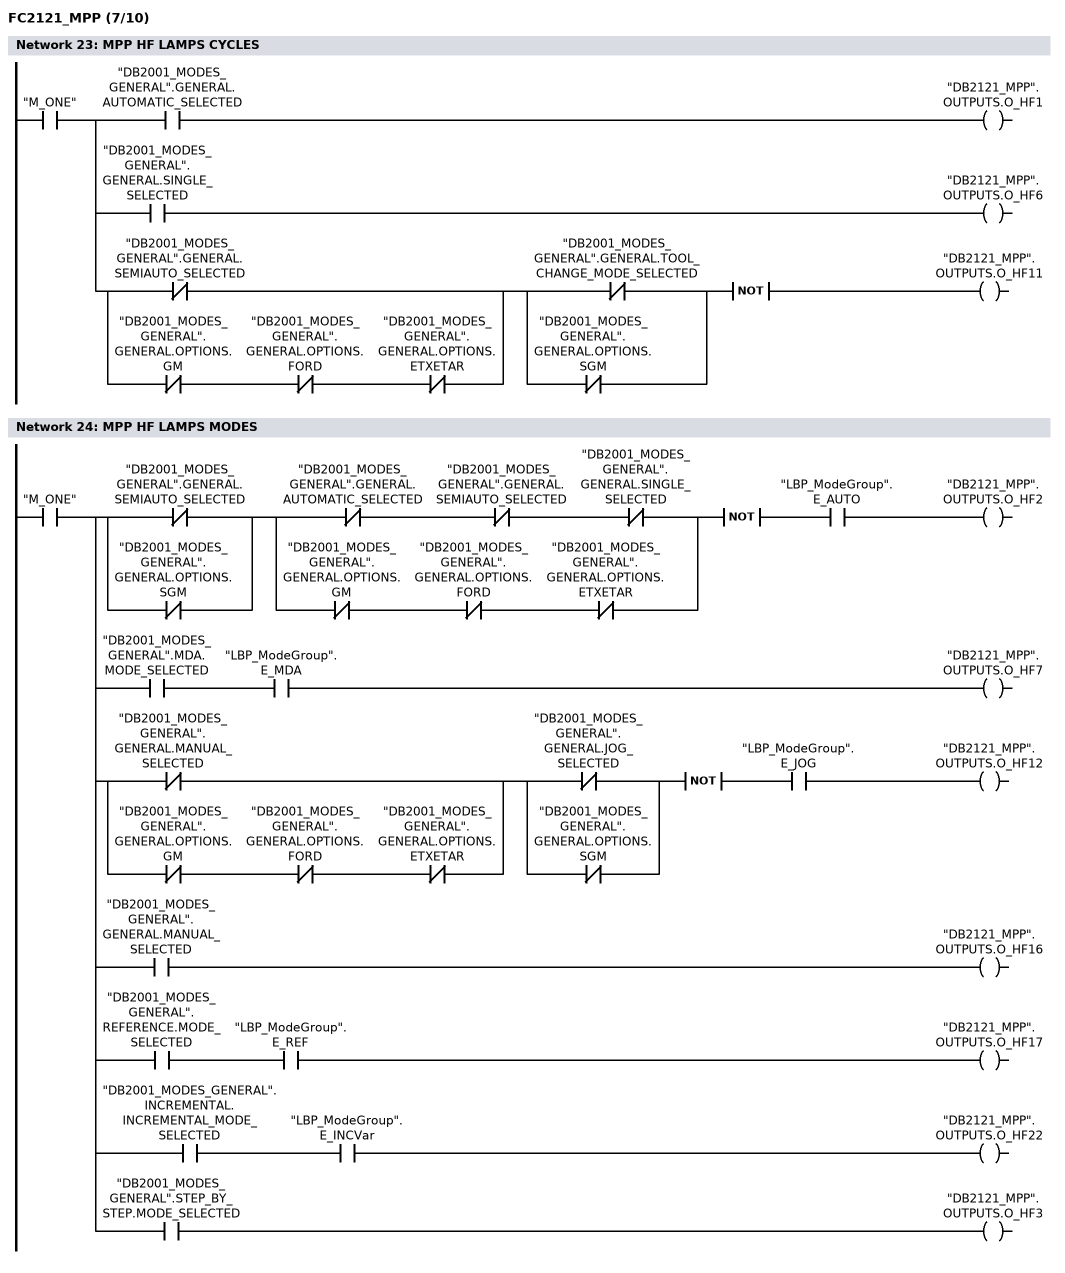
   RUNG wire#powerrail
      Contact( "M_ONE" )
      wire#w1
      Contact( "DB2001_MODES_GENERAL".GENERAL.AUTOMATIC_SELECTED )
      Coil( "DB2121_MPP".OUTPUTS.O_HF1 )
   END_RUNG
   RUNG wire#w1
      Contact( "DB2001_MODES_GENERAL".GENERAL.SINGLE_SELECTED )
      Coil( "DB2121_MPP".OUTPUTS.O_HF6 )
   END_RUNG
   RUNG wire#w1
      I_Contact( "DB2001_MODES_GENERAL".GENERAL.SEMIAUTO_SELECTED )
      wire#w2
      I_Contact( "DB2001_MODES_GENERAL".GENERAL.TOOL_CHANGE_MODE_SELECTED )
      wire#w3
      Not()
      Coil( "DB2121_MPP".OUTPUTS.O_HF11 )
   END_RUNG
   RUNG wire#w1
      I_Contact( "DB2001_MODES_GENERAL".GENERAL.OPTIONS.GM )
      I_Contact( "DB2001_MODES_GENERAL".GENERAL.OPTIONS.FORD )
      I_Contact( "DB2001_MODES_GENERAL".GENERAL.OPTIONS.ETXETAR )
   END_RUNG wire#w2
   RUNG wire#w2
      I_Contact( "DB2001_MODES_GENERAL".GENERAL.OPTIONS.SGM )
   END_RUNG wire#w3
   // the same network as SCL:
   "DB2121_MPP".OUTPUTS.O_HF1 := "M_ONE" AND "DB2001_MODES_GENERAL".GENERAL.AUTOMATIC_SELECTED;
   "DB2121_MPP".OUTPUTS.O_HF6 := "M_ONE" AND "DB2001_MODES_GENERAL".GENERAL.SINGLE_SELECTED;
   "DB2121_MPP".OUTPUTS.O_HF11 := NOT ("M_ONE" AND (NOT "DB2001_MODES_GENERAL".GENERAL.SEMIAUTO_SELECTED OR (NOT "DB2001_MODES_GENERAL".GENERAL.OPTIONS.GM AND NOT "DB2001_MODES_GENERAL".GENERAL.OPTIONS.FORD AND NOT "DB2001_MODES_GENERAL".GENERAL.OPTIONS.ETXETAR)) AND (NOT "DB2001_MODES_GENERAL".GENERAL.TOOL_CHANGE_MODE_SELECTED OR NOT "DB2001_MODES_GENERAL".GENERAL.OPTIONS.SGM));
END_REGION

REGION Network 24: MPP HF LAMPS MODES
   RUNG wire#powerrail
      Contact( "M_ONE" )
      wire#w1
      I_Contact( "DB2001_MODES_GENERAL".GENERAL.SEMIAUTO_SELECTED )
      wire#w2
      I_Contact( "DB2001_MODES_GENERAL".GENERAL.AUTOMATIC_SELECTED )
      I_Contact( "DB2001_MODES_GENERAL".GENERAL.SEMIAUTO_SELECTED )
      I_Contact( "DB2001_MODES_GENERAL".GENERAL.SINGLE_SELECTED )
      wire#w3
      Not()
      Contact( "LBP_ModeGroup".E_AUTO )
      Coil( "DB2121_MPP".OUTPUTS.O_HF2 )
   END_RUNG
   RUNG wire#w1
      I_Contact( "DB2001_MODES_GENERAL".GENERAL.OPTIONS.SGM )
   END_RUNG wire#w2
   RUNG wire#w2
      I_Contact( "DB2001_MODES_GENERAL".GENERAL.OPTIONS.GM )
      I_Contact( "DB2001_MODES_GENERAL".GENERAL.OPTIONS.FORD )
      I_Contact( "DB2001_MODES_GENERAL".GENERAL.OPTIONS.ETXETAR )
   END_RUNG wire#w3
   RUNG wire#w1
      Contact( "DB2001_MODES_GENERAL".MDA.MODE_SELECTED )
      Contact( "LBP_ModeGroup".E_MDA )
      Coil( "DB2121_MPP".OUTPUTS.O_HF7 )
   END_RUNG
   RUNG wire#w1
      I_Contact( "DB2001_MODES_GENERAL".GENERAL.MANUAL_SELECTED )
      wire#w4
      I_Contact( "DB2001_MODES_GENERAL".GENERAL.JOG_SELECTED )
      wire#w5
      Not()
      Contact( "LBP_ModeGroup".E_JOG )
      Coil( "DB2121_MPP".OUTPUTS.O_HF12 )
   END_RUNG
   RUNG wire#w1
      I_Contact( "DB2001_MODES_GENERAL".GENERAL.OPTIONS.GM )
      I_Contact( "DB2001_MODES_GENERAL".GENERAL.OPTIONS.FORD )
      I_Contact( "DB2001_MODES_GENERAL".GENERAL.OPTIONS.ETXETAR )
   END_RUNG wire#w4
   RUNG wire#w4
      I_Contact( "DB2001_MODES_GENERAL".GENERAL.OPTIONS.SGM )
   END_RUNG wire#w5
   RUNG wire#w1
      Contact( "DB2001_MODES_GENERAL".GENERAL.MANUAL_SELECTED )
      Coil( "DB2121_MPP".OUTPUTS.O_HF16 )
   END_RUNG
   RUNG wire#w1
      Contact( "DB2001_MODES_GENERAL".REFERENCE.MODE_SELECTED )
      Contact( "LBP_ModeGroup".E_REF )
      Coil( "DB2121_MPP".OUTPUTS.O_HF17 )
   END_RUNG
   RUNG wire#w1
      Contact( "DB2001_MODES_GENERAL".INCREMENTAL.INCREMENTAL_MODE_SELECTED )
      Contact( "LBP_ModeGroup".E_INCVar )
      Coil( "DB2121_MPP".OUTPUTS.O_HF22 )
   END_RUNG
   RUNG wire#w1
      Contact( "DB2001_MODES_GENERAL".STEP_BY_STEP.MODE_SELECTED )
      Coil( "DB2121_MPP".OUTPUTS.O_HF3 )
   END_RUNG
   // the same network as SCL:
   "DB2121_MPP".OUTPUTS.O_HF2 := NOT ("M_ONE" AND (NOT "DB2001_MODES_GENERAL".GENERAL.SEMIAUTO_SELECTED OR NOT "DB2001_MODES_GENERAL".GENERAL.OPTIONS.SGM) AND ((NOT "DB2001_MODES_GENERAL".GENERAL.AUTOMATIC_SELECTED AND NOT "DB2001_MODES_GENERAL".GENERAL.SEMIAUTO_SELECTED AND NOT "DB2001_MODES_GENERAL".GENERAL.SINGLE_SELECTED) OR (NOT "DB2001_MODES_GENERAL".GENERAL.OPTIONS.GM AND NOT "DB2001_MODES_GENERAL".GENERAL.OPTIONS.FORD AND NOT "DB2001_MODES_GENERAL".GENERAL.OPTIONS.ETXETAR))) AND "LBP_ModeGroup".E_AUTO;
   "DB2121_MPP".OUTPUTS.O_HF7 := "M_ONE" AND "DB2001_MODES_GENERAL".MDA.MODE_SELECTED AND "LBP_ModeGroup".E_MDA;
   "DB2121_MPP".OUTPUTS.O_HF12 := NOT ("M_ONE" AND (NOT "DB2001_MODES_GENERAL".GENERAL.MANUAL_SELECTED OR (NOT "DB2001_MODES_GENERAL".GENERAL.OPTIONS.GM AND NOT "DB2001_MODES_GENERAL".GENERAL.OPTIONS.FORD AND NOT "DB2001_MODES_GENERAL".GENERAL.OPTIONS.ETXETAR)) AND (NOT "DB2001_MODES_GENERAL".GENERAL.JOG_SELECTED OR NOT "DB2001_MODES_GENERAL".GENERAL.OPTIONS.SGM)) AND "LBP_ModeGroup".E_JOG;
   "DB2121_MPP".OUTPUTS.O_HF16 := "M_ONE" AND "DB2001_MODES_GENERAL".GENERAL.MANUAL_SELECTED;
   "DB2121_MPP".OUTPUTS.O_HF17 := "M_ONE" AND "DB2001_MODES_GENERAL".REFERENCE.MODE_SELECTED AND "LBP_ModeGroup".E_REF;
   "DB2121_MPP".OUTPUTS.O_HF22 := "M_ONE" AND "DB2001_MODES_GENERAL".INCREMENTAL.INCREMENTAL_MODE_SELECTED AND "LBP_ModeGroup".E_INCVar;
   "DB2121_MPP".OUTPUTS.O_HF3 := "M_ONE" AND "DB2001_MODES_GENERAL".STEP_BY_STEP.MODE_SELECTED;
END_REGION

REGION Network 25: MPP HF LAMPS - AXES
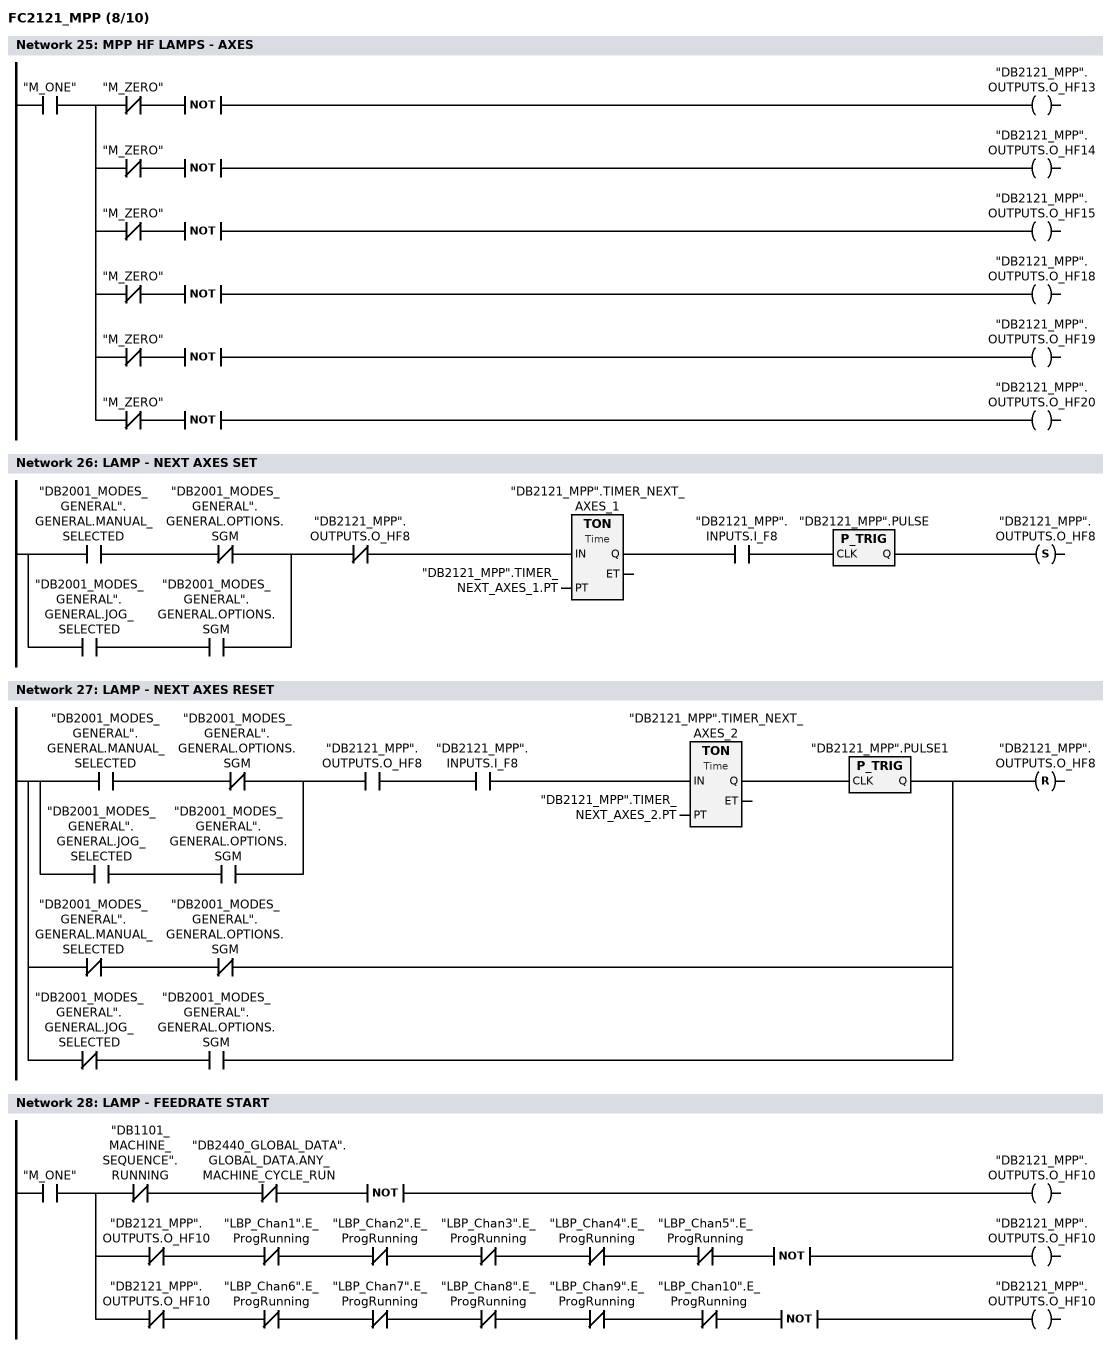
   RUNG wire#powerrail
      Contact( "M_ONE" )
      wire#w1
      I_Contact( "M_ZERO" )
      Not()
      Coil( "DB2121_MPP".OUTPUTS.O_HF13 )
   END_RUNG
   RUNG wire#w1
      I_Contact( "M_ZERO" )
      Not()
      Coil( "DB2121_MPP".OUTPUTS.O_HF14 )
   END_RUNG
   RUNG wire#w1
      I_Contact( "M_ZERO" )
      Not()
      Coil( "DB2121_MPP".OUTPUTS.O_HF15 )
   END_RUNG
   RUNG wire#w1
      I_Contact( "M_ZERO" )
      Not()
      Coil( "DB2121_MPP".OUTPUTS.O_HF18 )
   END_RUNG
   RUNG wire#w1
      I_Contact( "M_ZERO" )
      Not()
      Coil( "DB2121_MPP".OUTPUTS.O_HF19 )
   END_RUNG
   RUNG wire#w1
      I_Contact( "M_ZERO" )
      Not()
      Coil( "DB2121_MPP".OUTPUTS.O_HF20 )
   END_RUNG
   // the same network as SCL:
   "DB2121_MPP".OUTPUTS.O_HF13 := NOT ("M_ONE" AND NOT "M_ZERO");
   "DB2121_MPP".OUTPUTS.O_HF14 := NOT ("M_ONE" AND NOT "M_ZERO");
   "DB2121_MPP".OUTPUTS.O_HF15 := NOT ("M_ONE" AND NOT "M_ZERO");
   "DB2121_MPP".OUTPUTS.O_HF18 := NOT ("M_ONE" AND NOT "M_ZERO");
   "DB2121_MPP".OUTPUTS.O_HF19 := NOT ("M_ONE" AND NOT "M_ZERO");
   "DB2121_MPP".OUTPUTS.O_HF20 := NOT ("M_ONE" AND NOT "M_ZERO");
END_REGION

REGION Network 26: LAMP - NEXT AXES SET
   RUNG wire#powerrail
      Contact( "DB2001_MODES_GENERAL".GENERAL.MANUAL_SELECTED )
      I_Contact( "DB2001_MODES_GENERAL".GENERAL.OPTIONS.SGM )
      wire#w1
      I_Contact( "DB2121_MPP".OUTPUTS.O_HF8 )
      { S7_Templates := "time_type := Time" } "DB2121_MPP".TIMER_NEXT_AXES_1.TON(pt := "DB2121_MPP".TIMER_NEXT_AXES_1.PT, et =>)
      Contact( "DB2121_MPP".INPUTS.I_F8 )
      P_Trig( "DB2121_MPP".PULSE )
      S_Coil( "DB2121_MPP".OUTPUTS.O_HF8 )
   END_RUNG
   RUNG wire#powerrail
      Contact( "DB2001_MODES_GENERAL".GENERAL.JOG_SELECTED )
      Contact( "DB2001_MODES_GENERAL".GENERAL.OPTIONS.SGM )
   END_RUNG wire#w1
   // the same network as SCL:
   "DB2121_MPP".TIMER_NEXT_AXES_1.TON(IN := (("DB2001_MODES_GENERAL".GENERAL.MANUAL_SELECTED AND NOT "DB2001_MODES_GENERAL".GENERAL.OPTIONS.SGM) OR ("DB2001_MODES_GENERAL".GENERAL.JOG_SELECTED AND "DB2001_MODES_GENERAL".GENERAL.OPTIONS.SGM)) AND NOT "DB2121_MPP".OUTPUTS.O_HF8,
                           PT := "DB2121_MPP".TIMER_NEXT_AXES_1.PT);
   #_w1 := "DB2121_MPP".TIMER_NEXT_AXES_1.Q AND "DB2121_MPP".INPUTS.I_F8;
   #_w2 := #_w1 AND NOT "DB2121_MPP".PULSE;   // rising edge
   "DB2121_MPP".PULSE := #_w1;
   IF #_w2 THEN "DB2121_MPP".OUTPUTS.O_HF8 := TRUE; END_IF;
END_REGION

REGION Network 27: LAMP - NEXT AXES RESET
   RUNG wire#powerrail
      Contact( "DB2001_MODES_GENERAL".GENERAL.MANUAL_SELECTED )
      I_Contact( "DB2001_MODES_GENERAL".GENERAL.OPTIONS.SGM )
      wire#w1
      Contact( "DB2121_MPP".OUTPUTS.O_HF8 )
      Contact( "DB2121_MPP".INPUTS.I_F8 )
      { S7_Templates := "time_type := Time" } "DB2121_MPP".TIMER_NEXT_AXES_2.TON(pt := "DB2121_MPP".TIMER_NEXT_AXES_2.PT, et =>)
      P_Trig( "DB2121_MPP".PULSE1 )
      wire#w2
      R_Coil( "DB2121_MPP".OUTPUTS.O_HF8 )
   END_RUNG
   RUNG wire#powerrail
      Contact( "DB2001_MODES_GENERAL".GENERAL.JOG_SELECTED )
      Contact( "DB2001_MODES_GENERAL".GENERAL.OPTIONS.SGM )
   END_RUNG wire#w1
   RUNG wire#powerrail
      I_Contact( "DB2001_MODES_GENERAL".GENERAL.MANUAL_SELECTED )
      I_Contact( "DB2001_MODES_GENERAL".GENERAL.OPTIONS.SGM )
   END_RUNG wire#w2
   RUNG wire#powerrail
      I_Contact( "DB2001_MODES_GENERAL".GENERAL.JOG_SELECTED )
      Contact( "DB2001_MODES_GENERAL".GENERAL.OPTIONS.SGM )
   END_RUNG wire#w2
   // the same network as SCL:
   "DB2121_MPP".TIMER_NEXT_AXES_2.TON(IN := (("DB2001_MODES_GENERAL".GENERAL.MANUAL_SELECTED AND NOT "DB2001_MODES_GENERAL".GENERAL.OPTIONS.SGM) OR ("DB2001_MODES_GENERAL".GENERAL.JOG_SELECTED AND "DB2001_MODES_GENERAL".GENERAL.OPTIONS.SGM)) AND "DB2121_MPP".OUTPUTS.O_HF8 AND "DB2121_MPP".INPUTS.I_F8,
                           PT := "DB2121_MPP".TIMER_NEXT_AXES_2.PT);
   #_w1 := "DB2121_MPP".TIMER_NEXT_AXES_2.Q AND NOT "DB2121_MPP".PULSE1;   // rising edge
   "DB2121_MPP".PULSE1 := "DB2121_MPP".TIMER_NEXT_AXES_2.Q;
   IF #_w1 OR (NOT "DB2001_MODES_GENERAL".GENERAL.MANUAL_SELECTED AND NOT "DB2001_MODES_GENERAL".GENERAL.OPTIONS.SGM) OR (NOT "DB2001_MODES_GENERAL".GENERAL.JOG_SELECTED AND "DB2001_MODES_GENERAL".GENERAL.OPTIONS.SGM) THEN
       "DB2121_MPP".OUTPUTS.O_HF8 := FALSE;
   END_IF;
END_REGION

REGION Network 28: LAMP - FEEDRATE START
   RUNG wire#powerrail
      Contact( "M_ONE" )
      wire#w1
      I_Contact( "DB1101_MACHINE_SEQUENCE".RUNNING )
      I_Contact( "DB2440_GLOBAL_DATA".GLOBAL_DATA.ANY_MACHINE_CYCLE_RUN )
      Not()
      Coil( "DB2121_MPP".OUTPUTS.O_HF10 )
   END_RUNG
   RUNG wire#w1
      I_Contact( "DB2121_MPP".OUTPUTS.O_HF10 )
      I_Contact( "LBP_Chan1".E_ProgRunning )
      I_Contact( "LBP_Chan2".E_ProgRunning )
      I_Contact( "LBP_Chan3".E_ProgRunning )
      I_Contact( "LBP_Chan4".E_ProgRunning )
      I_Contact( "LBP_Chan5".E_ProgRunning )
      Not()
      Coil( "DB2121_MPP".OUTPUTS.O_HF10 )
   END_RUNG
   RUNG wire#w1
      I_Contact( "DB2121_MPP".OUTPUTS.O_HF10 )
      I_Contact( "LBP_Chan6".E_ProgRunning )
      I_Contact( "LBP_Chan7".E_ProgRunning )
      I_Contact( "LBP_Chan8".E_ProgRunning )
      I_Contact( "LBP_Chan9".E_ProgRunning )
      I_Contact( "LBP_Chan10".E_ProgRunning )
      Not()
      Coil( "DB2121_MPP".OUTPUTS.O_HF10 )
   END_RUNG
   // the same network as SCL:
   "DB2121_MPP".OUTPUTS.O_HF10 := NOT ("M_ONE" AND NOT "DB1101_MACHINE_SEQUENCE".RUNNING AND NOT "DB2440_GLOBAL_DATA".GLOBAL_DATA.ANY_MACHINE_CYCLE_RUN);
   "DB2121_MPP".OUTPUTS.O_HF10 := NOT ("M_ONE" AND NOT "DB2121_MPP".OUTPUTS.O_HF10 AND NOT "LBP_Chan1".E_ProgRunning AND NOT "LBP_Chan2".E_ProgRunning AND NOT "LBP_Chan3".E_ProgRunning AND NOT "LBP_Chan4".E_ProgRunning AND NOT "LBP_Chan5".E_ProgRunning);
   "DB2121_MPP".OUTPUTS.O_HF10 := NOT ("M_ONE" AND NOT "DB2121_MPP".OUTPUTS.O_HF10 AND NOT "LBP_Chan6".E_ProgRunning AND NOT "LBP_Chan7".E_ProgRunning AND NOT "LBP_Chan8".E_ProgRunning AND NOT "LBP_Chan9".E_ProgRunning AND NOT "LBP_Chan10".E_ProgRunning);
END_REGION

REGION Network 29: MPP HF LAMPS - NC START/STOP - FEEDRATE STOP
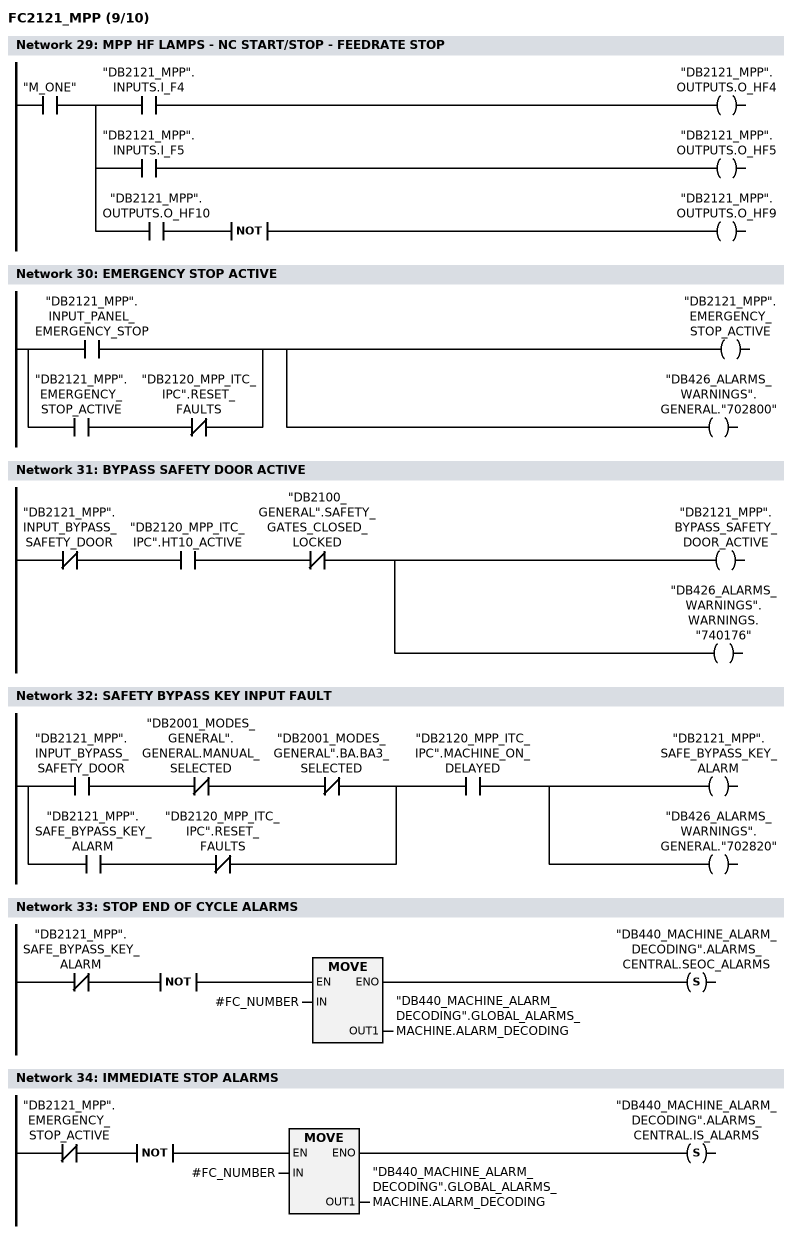
   RUNG wire#powerrail
      Contact( "M_ONE" )
      wire#w1
      Contact( "DB2121_MPP".INPUTS.I_F4 )
      Coil( "DB2121_MPP".OUTPUTS.O_HF4 )
   END_RUNG
   RUNG wire#w1
      Contact( "DB2121_MPP".INPUTS.I_F5 )
      Coil( "DB2121_MPP".OUTPUTS.O_HF5 )
   END_RUNG
   RUNG wire#w1
      Contact( "DB2121_MPP".OUTPUTS.O_HF10 )
      Not()
      Coil( "DB2121_MPP".OUTPUTS.O_HF9 )
   END_RUNG
   // the same network as SCL:
   "DB2121_MPP".OUTPUTS.O_HF4 := "M_ONE" AND "DB2121_MPP".INPUTS.I_F4;
   "DB2121_MPP".OUTPUTS.O_HF5 := "M_ONE" AND "DB2121_MPP".INPUTS.I_F5;
   "DB2121_MPP".OUTPUTS.O_HF9 := NOT ("M_ONE" AND "DB2121_MPP".OUTPUTS.O_HF10);
END_REGION

REGION Network 30: EMERGENCY STOP ACTIVE
   RUNG wire#powerrail
      Contact( "DB2121_MPP".INPUT_PANEL_EMERGENCY_STOP )
      wire#w1
      Coil( "DB2121_MPP".EMERGENCY_STOP_ACTIVE )
   END_RUNG
   RUNG wire#powerrail
      Contact( "DB2121_MPP".EMERGENCY_STOP_ACTIVE )
      I_Contact( "DB2120_MPP_ITC_IPC".RESET_FAULTS )
   END_RUNG wire#w1
   RUNG wire#w1
      Coil( "DB426_ALARMS_WARNINGS".GENERAL."702800" )
   END_RUNG
   // the same network as SCL:
   "DB2121_MPP".EMERGENCY_STOP_ACTIVE := "DB2121_MPP".INPUT_PANEL_EMERGENCY_STOP OR ("DB2121_MPP".EMERGENCY_STOP_ACTIVE AND NOT "DB2120_MPP_ITC_IPC".RESET_FAULTS);
   "DB426_ALARMS_WARNINGS".GENERAL."702800" := "DB2121_MPP".EMERGENCY_STOP_ACTIVE;
END_REGION

REGION Network 31: BYPASS SAFETY DOOR ACTIVE
   RUNG wire#powerrail
      I_Contact( "DB2121_MPP".INPUT_BYPASS_SAFETY_DOOR )
      Contact( "DB2120_MPP_ITC_IPC".HT10_ACTIVE )
      I_Contact( "DB2100_GENERAL".SAFETY_GATES_CLOSED_LOCKED )
      wire#w1
      Coil( "DB2121_MPP".BYPASS_SAFETY_DOOR_ACTIVE )
   END_RUNG
   RUNG wire#w1
      Coil( "DB426_ALARMS_WARNINGS".WARNINGS."740176" )
   END_RUNG
   // the same network as SCL:
   "DB2121_MPP".BYPASS_SAFETY_DOOR_ACTIVE := NOT "DB2121_MPP".INPUT_BYPASS_SAFETY_DOOR AND "DB2120_MPP_ITC_IPC".HT10_ACTIVE AND NOT "DB2100_GENERAL".SAFETY_GATES_CLOSED_LOCKED;
   "DB426_ALARMS_WARNINGS".WARNINGS."740176" := "DB2121_MPP".BYPASS_SAFETY_DOOR_ACTIVE;
END_REGION

REGION Network 32: SAFETY BYPASS KEY INPUT FAULT
   RUNG wire#powerrail
      Contact( "DB2121_MPP".INPUT_BYPASS_SAFETY_DOOR )
      I_Contact( "DB2001_MODES_GENERAL".GENERAL.MANUAL_SELECTED )
      I_Contact( "DB2001_MODES_GENERAL".BA.BA3_SELECTED )
      wire#w1
      Contact( "DB2120_MPP_ITC_IPC".MACHINE_ON_DELAYED )
      wire#w2
      Coil( "DB2121_MPP".SAFE_BYPASS_KEY_ALARM )
   END_RUNG
   RUNG wire#powerrail
      Contact( "DB2121_MPP".SAFE_BYPASS_KEY_ALARM )
      I_Contact( "DB2120_MPP_ITC_IPC".RESET_FAULTS )
   END_RUNG wire#w1
   RUNG wire#w2
      Coil( "DB426_ALARMS_WARNINGS".GENERAL."702820" )
   END_RUNG
   // the same network as SCL:
   "DB2121_MPP".SAFE_BYPASS_KEY_ALARM := (("DB2121_MPP".INPUT_BYPASS_SAFETY_DOOR AND NOT "DB2001_MODES_GENERAL".GENERAL.MANUAL_SELECTED AND NOT "DB2001_MODES_GENERAL".BA.BA3_SELECTED) OR ("DB2121_MPP".SAFE_BYPASS_KEY_ALARM AND NOT "DB2120_MPP_ITC_IPC".RESET_FAULTS)) AND "DB2120_MPP_ITC_IPC".MACHINE_ON_DELAYED;
   "DB426_ALARMS_WARNINGS".GENERAL."702820" := "DB2121_MPP".SAFE_BYPASS_KEY_ALARM;
END_REGION

REGION Network 33: STOP END OF CYCLE ALARMS
   RUNG wire#powerrail
      I_Contact( "DB2121_MPP".SAFE_BYPASS_KEY_ALARM )
      Not()
      { S7_GenerateENO := "TRUE" } Move(in := #FC_NUMBER, out1 => "DB440_MACHINE_ALARM_DECODING".GLOBAL_ALARMS_MACHINE.ALARM_DECODING)
      S_Coil( "DB440_MACHINE_ALARM_DECODING".ALARMS_CENTRAL.SEOC_ALARMS )
   END_RUNG
   // the same network as SCL:
   // ENO of a box is taken as its EN; it also drops when the box reports an error
   IF NOT (NOT "DB2121_MPP".SAFE_BYPASS_KEY_ALARM) THEN
       "DB440_MACHINE_ALARM_DECODING".GLOBAL_ALARMS_MACHINE.ALARM_DECODING := #FC_NUMBER;
       "DB440_MACHINE_ALARM_DECODING".ALARMS_CENTRAL.SEOC_ALARMS := TRUE;
   END_IF;
END_REGION

REGION Network 34: IMMEDIATE STOP ALARMS
   RUNG wire#powerrail
      I_Contact( "DB2121_MPP".EMERGENCY_STOP_ACTIVE )
      Not()
      { S7_GenerateENO := "TRUE" } Move(in := #FC_NUMBER, out1 => "DB440_MACHINE_ALARM_DECODING".GLOBAL_ALARMS_MACHINE.ALARM_DECODING)
      S_Coil( "DB440_MACHINE_ALARM_DECODING".ALARMS_CENTRAL.IS_ALARMS )
   END_RUNG
   // the same network as SCL:
   // ENO of a box is taken as its EN; it also drops when the box reports an error
   IF NOT (NOT "DB2121_MPP".EMERGENCY_STOP_ACTIVE) THEN
       "DB440_MACHINE_ALARM_DECODING".GLOBAL_ALARMS_MACHINE.ALARM_DECODING := #FC_NUMBER;
       "DB440_MACHINE_ALARM_DECODING".ALARMS_CENTRAL.IS_ALARMS := TRUE;
   END_IF;
END_REGION

REGION Network 35: WARNING
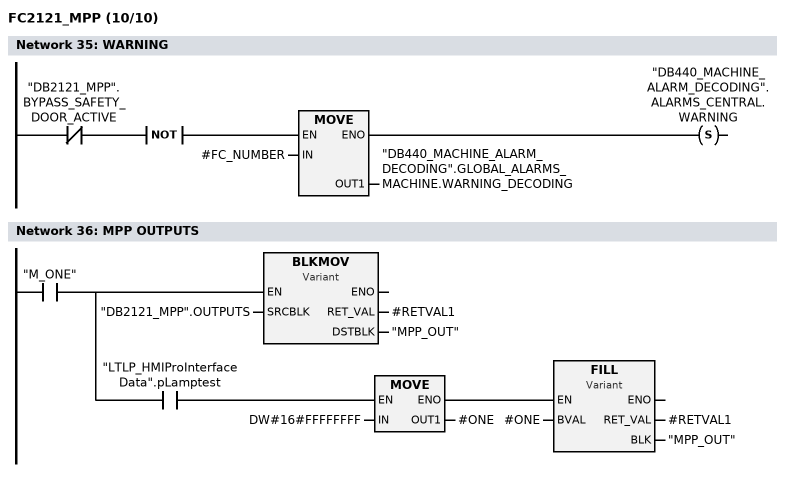
   RUNG wire#powerrail
      I_Contact( "DB2121_MPP".BYPASS_SAFETY_DOOR_ACTIVE )
      Not()
      { S7_GenerateENO := "TRUE" } Move(in := #FC_NUMBER, out1 => "DB440_MACHINE_ALARM_DECODING".GLOBAL_ALARMS_MACHINE.WARNING_DECODING)
      S_Coil( "DB440_MACHINE_ALARM_DECODING".ALARMS_CENTRAL.WARNING )
   END_RUNG
   // the same network as SCL:
   // ENO of a box is taken as its EN; it also drops when the box reports an error
   IF NOT (NOT "DB2121_MPP".BYPASS_SAFETY_DOOR_ACTIVE) THEN
       "DB440_MACHINE_ALARM_DECODING".GLOBAL_ALARMS_MACHINE.WARNING_DECODING := #FC_NUMBER;
       "DB440_MACHINE_ALARM_DECODING".ALARMS_CENTRAL.WARNING := TRUE;
   END_IF;
END_REGION

REGION Network 36: MPP OUTPUTS
   RUNG wire#powerrail
      Contact( "M_ONE" )
      wire#w1
      { S7_Templates := "blk_type := Variant" } BLKMOV(SRCBLK := "DB2121_MPP".OUTPUTS, RET_VAL => #RETVAL1, DSTBLK => "MPP_OUT")
   END_RUNG
   RUNG wire#w1
      Contact( "LTLP_HMIProInterfaceData".pLamptest )
      { S7_GenerateENO := "TRUE" } Move(in := DW#16#FFFFFFFF, out1 => #ONE)
      { S7_Templates := "ptr_type := Variant" } FILL(BVAL := #ONE, RET_VAL => #RETVAL1, BLK => "MPP_OUT")
   END_RUNG
   // the same network as SCL:
   // ENO of a box is taken as its EN; it also drops when the box reports an error
   #_w1 := "M_ONE";
   IF #_w1 THEN #RETVAL1 := BLKMOV(SRCBLK := "DB2121_MPP".OUTPUTS, DSTBLK => "MPP_OUT"); END_IF;
   IF #_w1 AND "LTLP_HMIProInterfaceData".pLamptest THEN
       #ONE := DW#16#FFFFFFFF;
       #RETVAL1 := FILL(BVAL := #ONE, BLK => "MPP_OUT");
   END_IF;
END_REGION
END_FUNCTION
